(* CoDeSys 2.3.9.42 project: komp_new.pro *)
(* Libraries: Standard.lib 2.12.10 17:48:34, SYSLIBCALLBACK.LIB 2.12.10 17:48:32 *)

(* PLC configuration (modules and I/O channels)
S4_1 AT %IX12.0 [BOOLOnX_I] Ch_1 Digital input
S4_2 AT %IX12.1 [BOOLOnX_I] Ch_2 Digital input
S5_1 AT %IX12.2 [BOOLOnX_I] Ch_3 Digital input
S5_2 AT %IX12.3 [BOOLOnX_I] Ch_4 Digital input
S6_1 AT %IX12.4 [BOOLOnX_I] Ch_5 Digital input
S6_2 AT %IX12.5 [BOOLOnX_I] Ch_6 Digital input
S7_1 AT %IX12.6 [BOOLOnX_I] Ch_7 Digital input
S7_2 AT %IX12.7 [BOOLOnX_I] Ch_8 Digital input
S8_1 AT %IX12.8 [BOOLOnX_I] Ch_9 Digital input
S8_2 AT %IX12.9 [BOOLOnX_I] Ch_10 Digital input
S9_1 AT %IX12.10 [BOOLOnX_I] Ch_11 Digital input
S9_2 AT %IX12.11 [BOOLOnX_I] Ch_12 Digital input
S10_1 AT %IX12.12 [BOOLOnX_I] Ch_13 Digital input
S10_2 AT %IX12.13 [BOOLOnX_I] Ch_14 Digital input
S11_1 AT %IX12.14 [BOOLOnX_I] Ch_15 Digital input
S11_2 AT %IX12.15 [BOOLOnX_I] Ch_16 Digital input
S14_1 AT %IX13.0 [BOOLOnX_I] Ch_1 Digital input
S14_2 AT %IX13.1 [BOOLOnX_I] Ch_2 Digital input
S18_1 AT %IX13.2 [BOOLOnX_I] Ch_3 Digital input
S18_2 AT %IX13.3 [BOOLOnX_I] Ch_4 Digital input
S19_1 AT %IX13.4 [BOOLOnX_I] Ch_5 Digital input
S19_2 AT %IX13.5 [BOOLOnX_I] Ch_6 Digital input
_controlFazaDI AT %IX13.6 [BOOLOnX_I] Ch_7 Digital input
_currentHighJD5DI AT %IX13.7 [BOOLOnX_I] Ch_8 Digital input
_vacumContactOnDI AT %IX13.8 [BOOLOnX_I] Ch_9 Digital input
_vacumContactOffDI AT %IX13.9 [BOOLOnX_I] Ch_10 Digital input
__1pressLevelInDI AT %IX13.10 [BOOLOnX_I] Ch_11 Digital input
__2pressLevelInDI AT %IX13.11 [BOOLOnX_I] Ch_12 Digital input
__3pressLevelInDI AT %IX13.12 [BOOLOnX_I] Ch_13 Digital input
__4pressLevelInDI AT %IX13.13 [BOOLOnX_I] Ch_14 Digital input
_4pressLeveOutDI AT %IX13.14 [BOOLOnX_I] Ch_15 Digital input
pressWaterDI AT %IX13.15 [BOOLOnX_I] Ch_16 Digital input
KM4_1 AT %QX0.0 [BOOLOnX_Q] Ch_1 Digital output
KM4_2 AT %QX0.1 [BOOLOnX_Q] Ch_2 Digital output
KM5_1 AT %QX0.2 [BOOLOnX_Q] Ch_3 Digital output
KM5_2 AT %QX0.3 [BOOLOnX_Q] Ch_4 Digital output
KM6_1 AT %QX0.4 [BOOLOnX_Q] Ch_5 Digital output
KM6_2 AT %QX0.5 [BOOLOnX_Q] Ch_6 Digital output
KM7_1 AT %QX0.6 [BOOLOnX_Q] Ch_7 Digital output
KM7_2 AT %QX0.7 [BOOLOnX_Q] Ch_8 Digital output
KM8_1 AT %QX0.8 [BOOLOnX_Q] Ch_9 Digital output
KM8_2 AT %QX0.9 [BOOLOnX_Q] Ch_10 Digital output
KM9_1 AT %QX0.10 [BOOLOnX_Q] Ch_11 Digital output
KM9_2 AT %QX0.11 [BOOLOnX_Q] Ch_12 Digital output
KM10_1 AT %QX0.12 [BOOLOnX_Q] Ch_13 Digital output
KM10_2 AT %QX0.13 [BOOLOnX_Q] Ch_14 Digital output
KM11_1 AT %QX0.14 [BOOLOnX_Q] Ch_15 Digital output
KM11_2 AT %QX0.15 [BOOLOnX_Q] Ch_16 Digital output
KM14_1 AT %QX1.0 [BOOLOnX_Q] Ch_1 Digital output
KM14_2 AT %QX1.1 [BOOLOnX_Q] Ch_2 Digital output
KM18_1 AT %QX1.2 [BOOLOnX_Q] Ch_3 Digital output
KM18_2 AT %QX1.3 [BOOLOnX_Q] Ch_4 Digital output
readyWater AT %QX1.4 [BOOLOnX_Q] Ch_5 Digital output
readyOil AT %QX1.5 [BOOLOnX_Q] Ch_6 Digital output
_oilGate_1 AT %QX1.6 [BOOLOnX_Q] Ch_7 Digital output
_oilGate_2 AT %QX1.7 [BOOLOnX_Q] Ch_8 Digital output
KM2 AT %QX1.8 [BOOLOnX_Q] Ch_9 Digital output
_rejimModeDO AT %QX1.9 [BOOLOnX_Q] Ch_10 Digital output
KM1 AT %QX1.10 [BOOLOnX_Q] Ch_11 Digital output
_PuskModeDO AT %QX1.11 [BOOLOnX_Q] Ch_12 Digital output
_kompOnDO AT %QX1.12 [BOOLOnX_Q] Ch_13 Digital output
_kompOffDO AT %QX1.13 [BOOLOnX_Q] Ch_14 Digital output
_alarmLedDO_blink AT %QX1.14 [BOOLOnX_Q] Ch_15 Digital output
_stopModeDO AT %QX1.15 [BOOLOnX_Q] Ch_16 Digital output
AT %IW0 [WORDOnW_I] Ch_1 Input word
AT %IW1 [WORDOnW_I] Ch_2 Input word
AT %IW2 [WORDOnW_I] Ch_3 Input word
AT %IW3 [WORDOnW_I] Ch_4 Input word
AT %IW4 [WORDOnW_I] Ch_1 Input word
AT %IW5 [WORDOnW_I] Ch_2 Input word
AT %IW6 [WORDOnW_I] Ch_3 Input word
AT %IW7 [WORDOnW_I] Ch_4 Input word
AT %IW8 [WORDOnW_I] Ch_1 Input word
AT %IW9 [WORDOnW_I] Ch_2 Input word
AT %IW10 [WORDOnW_I] Ch_3 Input word
AT %IW11 [WORDOnW_I] Ch_4 Input word
_konsovikMechanikMotor AT %IX14.0 [BOOLOnX_I] Ch_1 Digital input
_emergencyStop AT %IX14.1 [BOOLOnX_I] Ch_2 Digital input
_buttonStop AT %IX14.2 [BOOLOnX_I] Ch_3 Digital input
_buttonRejim AT %IX14.3 [BOOLOnX_I] Ch_4 Digital input
_buttonPusk AT %IX14.4 [BOOLOnX_I] Ch_5 Digital input
_switchAuto AT %IX14.5 [BOOLOnX_I] Ch_6 Digital input
_switchManual AT %IX14.6 [BOOLOnX_I] Ch_7 Digital input
_emergencyStopMashZal AT %IX14.7 [BOOLOnX_I] Ch_8 Digital input
gazaAnalizMashzal AT %IX14.8 [BOOLOnX_I] Ch_9 Digital input
gazaAnaliz AT %IX14.9 [BOOLOnX_I] Ch_10 Digital input
_pressOilMINDI AT %IX14.10 [BOOLOnX_I] Ch_11 Digital input
_pressOilMAXDI AT %IX14.11 [BOOLOnX_I] Ch_12 Digital input
pressOil_DI AT %IX14.12 [BOOLOnX_I] Ch_13 Digital input
AT %IX14.13 [BOOLOnX_I] Ch_14 Digital input
AT %IX14.14 [BOOLOnX_I] Ch_15 Digital input
AT %IX14.15 [BOOLOnX_I] Ch_16 Digital input
Fieldbus variables [FB_VARS] node 1, in %IB0 out %QB0
Flag variables [FLAG_VARS] node 2, in %IB0 out %QB0
*)

(* Global variable list: _L *)
VAR_GLOBAL
	L11_PUSK : BOOL;
	L12_PUSK : BOOL;
	TO_LIST13: BOOL;

END_VAR

(* Global variable list: _S *)
VAR_GLOBAL
	_17S_1: BOOL;
	_16S_1: BOOL;
END_VAR

(* Global variable list: Global_Variables *)
VAR_GLOBAL
	_alarmLedDO : BOOL;
	alarm : ALARMS;
	_pressWaterDI : BOOL;
	_pressOil_DI : BOOL;
	_1pressLevelInDI : BOOL;
	_2pressLevelInDI : BOOL;
	_3pressLevelInDI : BOOL;
	_4pressLevelInDI : BOOL;
	(*waterPump1 : Pumps;
	waterPump2 : Pumps;
	oilPump1 : Pumps;
	oilPump2 : Pumps;
	_18gate : GateValve;
	_4gate : GateValve;
	_5gate : GateValve;
	_6gate : GateValve;
	_7gate : GateValve;
	_8gate : GateValve;
	_9gate : GateValve;
	_10gate : GateValve;
	_11gate : GateValve;
	_14gate : GateValve;
	_17gate : GateValve;
	_19gate : GateValve;
	_20gate : GateValve;
	heater : Heaters;
	komp : Compressor;

	wtrTimeWORD AT %QW256: WORD := 2;
	oilTimeWORD  AT %QW257: WORD := 2;

	MODE AT %QW280 : WORD;

	gate18TimeWORD  AT %IW258 :WORD := 2;
	gate4TimeWORD  AT %IW259 :WORD := 2;
	gate5TimeWORD  AT %IW260 :WORD := 2;
	gate6TimeWORD  AT %IW261 :WORD := 2;
	gate7TimeWORD  AT %IW262 :WORD := 2;
	gate8TimeWORD  AT %IW263 :WORD := 2;
	gate9TimeWORD  AT %IW264 :WORD := 2;
	gate10TimeWORD  AT %IW265 :WORD := 2;
	gate11TimeWORD  AT %IW266 :WORD := 2;
	gate14TimeWORD  AT %IW267 :WORD := 2;
	gate17TimeWORD  AT %QW268 :WORD := 2;
	gate17T3  AT %IW268 :WORD := 3;
	gate17T4  AT %MW268 :WORD := 4;
	
	wtrTime : TIME := T#2s;
	oilTime : TIME := T#2s;
	gate18Time  :TIME := T#2s;
	gate4Time  :TIME := T#2s;
	gate5Time  :TIME := T#2s;
	gate6Time  :TIME := T#2s;
	gate7Time  :TIME := T#2s;
	gate8Time  :TIME := T#2s;
	gate9Time  :TIME := T#2s;
	gate10Time :TIME := T#2s;
	gate11Time  :TIME := T#2s;
	gate14Time  :TIME := T#2s;
	gate17Time  :TIME := T#2s;

	goRejim AT %QX269.0 : BOOL;
	goPusk AT %QX269.1: BOOL;
	goSTOP AT %QX269.2 : BOOL;
	kompReady AT %QX269.3 : BOOL := FALSE;
	isOK AT %QX269.4: BOOL := TRUE;

	_4gate_open  AT %IX269.5 : BOOL;
	_4gate_close  AT %IX269.6 : BOOL;
	_5gate_open  AT %IX269.7 : BOOL;
	_5gate_close  AT %IX269.8 : BOOL;
	_6gate_open  AT %IX269.9 : BOOL;
	_6gate_close  AT %IX269.10 : BOOL;
	_7gate_open  AT %IX269.11 : BOOL;
	_7gate_close  AT %IX269.12 : BOOL;
	_8gate_open  AT %IX269.13 : BOOL;
	_8gate_close  AT %IX269.14 : BOOL;
	_9gate_open  AT %IX269.15 : BOOL;
	_9gate_close  AT %IX270.0 : BOOL;
	_10gate_open  AT %IX270.1 : BOOL;
	_10gate_close  AT %IX270.2 : BOOL;
	_11gate_open  AT %IX270.3 : BOOL;
	_11gate_close  AT %IX270.4 : BOOL;
	_14gate_open  AT %IX270.5 : BOOL;
	_14gate_close  AT %IX270.6 : BOOL;
	_18gate_open  AT %IX270.7 : BOOL;
	_18gate_close  AT %IX270.8 : BOOL;
	_19gate_open  AT %IX270.9 : BOOL;
	_19gate_close  AT %IX270.10 : BOOL;
	_20gate_open  AT %IX270.11 : BOOL;
	_20gate_close  AT %IX270.12 : BOOL;
	oilPump1_run  AT %IX270.13 : BOOL;
	oilPump2_run  AT %IX270.14 : BOOL;
	waterPump1_run  AT %IX270.15 : BOOL;
	waterPump2_run  AT %IX271.0 : BOOL;
	komp_run  AT %IX271.1 : BOOL;
	komp_stop  AT %IX271.2 : BOOL;
	autoManual  AT %IX272.0 : BOOL;
	*)


END_VAR

(* Global variable list: K *)
VAR_GLOBAL

	K01: BOOL;
	K1: BOOL;
	K2: BOOL;
	K3: BOOL;
	K4: BOOL;
	K5: BOOL;
	K6 : BOOL;
	K7 : BOOL;
	K8 : BOOL;
	K13 : BOOL;
	K14: BOOL;
	K15: BOOL;
END_VAR

(* Global variable list: KM *)
VAR_GLOBAL

	TRM7: BOOL := TRUE;
	KM3: BOOL; (*Nagrev gaza*)
(*
	KM1: BOOL; (* suv nasos*)
	KM2: BOOL; (*maslo nasos*)
	
	KM4_1: BOOL;  (*Zadvijka 4 katushka ochish*)
	KM4_2: BOOL;  (*Zadvijka 4 katushka YOPISH*)
	KM5_1: BOOL;  (*Zadvijka 5 katushka ochish*)
	KM5_2: BOOL;  (*Zadvijka 5 katushka ochish*)
	KM6_1 : BOOL; (*Zadvijka 6 katushka ochish*)
	KM6_2 : BOOL; (*Zadvijka 6 katushka YOPISH*)
	KM7_1: BOOL; (*Zadvijka 7 katushka ochish*)
	KM7_2: BOOL;  (*Zadvijka 7 katushka YOPISH*)
	KM8_1: BOOL; (*Zadvijka 8 katushka ochish*)
	KM8_2: BOOL; (*Zadvijka 8 katushka YOPISH*)
	KM9_1: BOOL;  (*Zadvijka 9 katushka ochish*)
	KM9_2: BOOL;  (*Zadvijka 9 katushka YOPISH*)
	KM10_1: BOOL;  (*Zadvijka 10 katushka ochish*)
	KM10_2: BOOL; (*Zadvijka 10 katushka YOPISH*)
	KM11_1: BOOL; (*Zadvijka 11 katushka ochish*)
	KM11_2: BOOL; (*Zadvijka 11 katushka YOPISH*)
	KM13_1: BOOL;  (*Zadvijka 13 katushka ochish*)
	KM13_2: BOOL; (*Zadvijka 13 katushka YOPISH*)
	KM14_1: BOOL;  (*Zadvijka 14 katushka ochish*)
	KM14_2: BOOL;  (*Zadvijka 14 katushka YOPISH*)
	KM15_1 : BOOL;  (*Zadvijka 15 katushka ochish*)
	KM15_2 : BOOL; (*Zadvijka 15 katushka YOPISH*)
	
	KM18_1 : BOOL; (*Zadvijka 18 katushka ochish*)
	KM18_2 : BOOL;	(*Zadvijka 18 katushka YOPISH*)
*)
	KM16_1: BOOL;  (*Zadvijka 16 katushka ochish*)
	KM16_2: BOOL; (*Zadvijka 16 katushka YOPISH*)
	KM17_1: BOOL; (*Zadvijka 17 katushka ochish*)
	KM17_2: BOOL; (*Zadvijka 17 katushka YOPISH*)
END_VAR

(* Global variable list: P *)
VAR_GLOBAL

	P0: BOOL;

	P1 : BOOL; 	(*GOTOVNOST*)
	P2 : BOOL; 	(*REJIM*)
	P3: BOOL; 	(* STOP kompressor*)
	P4 : BOOL;
	P5 : BOOL;
	P6 : BOOL;	 (* EKM vodinoy nasos*)
	P7 : BOOL; 	(* EKM maslo nasos*)


END_VAR

(* Global variable list: RV *)
VAR_GLOBAL


	RV3: BOOL;
	RV4: BOOL;
	RV5: BOOL;
	RV13: BOOL;
	RV15: BOOL;

	RV3TON: TON;
	RV4TON: TON;
	RV5TON: TON;
	RV13TON : TON;
	RV15TON : TON;


END_VAR

(* Global variable list: V_MODBUS *)
VAR_GLOBAL

	S4_1MB AT %MX100.0 : BOOL;
	S4_2MB AT %MX100.1 : BOOL;
	S5_1MB AT %MX100.2 : BOOL;
	S5_2MB AT %MX100.3 : BOOL;
	S6_1MB AT %MX100.4 : BOOL;
	S6_2MB AT %MX100.5 : BOOL;
	S7_1MB AT %MX100.6 : BOOL;
	S7_2MB AT %MX100.7 : BOOL;
	S8_1MB AT %MX100.8 : BOOL;
	S8_2MB AT %MX100.9 : BOOL;
	S9_1MB AT %MX100.10 : BOOL;
	S9_2MB AT %MX100.11 : BOOL;
	S10_1MB AT %MX100.12 : BOOL;
	S10_2MB AT %MX100.13 : BOOL;
	S11_1MB AT %MX100.14 : BOOL;
	S11_2MB AT %MX100.15 : BOOL;
	S14_1MB AT %MX101.0 : BOOL;
	S14_2MB AT %MX101.1 : BOOL;
	S18_1MB AT %MX101.2 : BOOL;
	S18_2MB AT %MX101.3 : BOOL;
	S19_1MB AT %MX101.4 : BOOL;
	S19_2MB AT %MX101.5 : BOOL;
	controlFazaDIMB AT %MX101.6 : BOOL;
	currentHighJD5DIMB AT %MX101.7 : BOOL;
	vacumContactOnDIMB AT %MX101.8 : BOOL;
	vacumContactOffDIMB AT %MX101.9 : BOOL;
	press1LevelInDIMB AT %MX101.10 : BOOL;
	press2LevelInDIMB AT %MX101.11 : BOOL;
	press3LevelInDIMB AT  %MX101.12 : BOOL;
	press4LevelInDIMB AT %MX101.13 : BOOL;
	press4LevelOutDIMB AT %MX101.14 : BOOL;
	pressWaterDIMB AT  %MX101.15 : BOOL;
	KM4_1MB AT %MX102.0 : BOOL;
	KM4_2MB AT %MX102.1 : BOOL;
	KM5_1MB AT %MX102.2 : BOOL;
	KM5_2MB AT %MX102.3 : BOOL;
	KM6_1MB AT %MX102.4 : BOOL;
	KM6_2MB AT %MX102.5 : BOOL;
	KM7_1MB AT %MX102.6 : BOOL;
	KM7_2MB AT %MX102.7 : BOOL;
	KM8_1MB AT %MX102.8 : BOOL;
	KM8_2MB AT %MX102.9 : BOOL;
	KM9_1MB AT %MX102.10 : BOOL;
	KM9_2MB AT %MX102.11 : BOOL;
	KM10_1MB AT %MX102.12 : BOOL;
	KM10_2MB AT %MX102.13 : BOOL;
	KM11_1MB AT %MX102.14 : BOOL;
	KM11_2MB AT %MX102.15 : BOOL;

	KM14_1MB AT %MX103.0 : BOOL;
	KM14_2MB AT %MX103.1 : BOOL;
	KM18_1MB AT %MX103.2 : BOOL;
	KM18_2MB AT %MX103.3 : BOOL;
	KM19_1MB AT %MX103.4 : BOOL;
	KM19_2MB AT %MX103.5 : BOOL;
	KM1_MB AT %MX103.6 : BOOL;
	KM2_MB AT %MX103.7 : BOOL;
	kompOnDO_MB AT %MX103.8 : BOOL;
	kompOffDO_MB AT %MX103.9 : BOOL;
	alarmLedDO_MB AT %MX103.10 : BOOL;
	stopModeDO_MB AT %MX103.11 : BOOL;
	acknowledgment_MB AT %MX103.12 : BOOL;
	gazaAnaliz_MB AT %MX103.12 : BOOL;
	gazaAnalizMashzal_MB  AT %MX103.13 : BOOL;
	serviceMODE_MB AT %MX103.14 : BOOL;
	SB3 AT %MX104.0: BOOL;  (*PUSK VODA knopka*)
	SB4 AT %MX104.1: BOOL;  (*STOP VODA knopka*)
	SB5 AT %MX104.2: BOOL; (*PUSK MASLO knopka*)
	SB6 AT %MX104.3: BOOL; (*STOP MASLO knopka*)
	SB7 AT %MX104.4: BOOL; (*PUSK NAGREV knopka*)
	SB8 AT %MX104.5: BOOL; (*STOP NAGREV knopka*)
	SB9 AT %MX104.6: BOOL; (*Zadvijka 4 ochish knopka*)
	SB10 AT %MX104.7: BOOL;  (*Zadvijka  4  YOPISH   knopka*)
	SB11 AT %MX104.8: BOOL; (*Zadvijka 5 ochish knopka*)
	SB12 AT %MX104.9: BOOL; (*Zadvijka 5 YOPISH knopka*)
	SB13 AT %MX104.10: BOOL; (*Zadvijka 6 ochish knopka*)
	SB14 AT %MX104.11: BOOL;  (*Zadvijka 6 YOPISH knopka*)
	SB15 AT %MX104.12: BOOL;  (*Zadvijka 7 ochish knopka*)
	SB16 AT %MX104.13: BOOL; (*Zadvijka 7 YOPISH knopka*)
	SB17 AT %MX104.14: BOOL;  (*Zadvijka 8 ochish knopka*)
	SB18 AT %MX104.15: BOOL; (*Zadvijka 8 YOPISH knopka*)

	SB19 AT %MX105.0: BOOL;	 (*Zadvijka 9 ochish knopka*)
	SB20 AT %MX105.1: BOOL;  (*Zadvijka 9 YOPISH knopka*)
	SB21 AT %MX105.2: BOOL;	 (*Zadvijka 10 ochish knopka*)
	SB22 AT %MX105.3: BOOL; (*Zadvijka 10 YOPISH knopka*)
	SB23 AT %MX105.4: BOOL; (*Zadvijka 11 ochish knopka*)
	SB24 AT %MX105.5: BOOL; (*Zadvijka 11 YOPISH knopka*)
	SB25 AT %MX105.6: BOOL;  (*Zadvijka 14 ochish knopka*)
	SB26 AT %MX105.7: BOOL;  (*Zadvijka 14 YOPISH knopka*)
	SB29 AT %MX105.8: BOOL;  (*Zadvijka 18 ochish knopka*)
	SB30 AT %MX105.9: BOOL;   (*Zadvijka 18 YOPISH knopka*)
	SB32 AT %MX105.10: BOOL; (*Zadvijka 16 YOPISH knopka*)
	SBA41 AT %IX14.12: BOOL; (* Avariyniy stop*)
	SBA41_MB AT %MX105.11: BOOL; (* Avariyniy stop*)
	SB42 AT  %IX14.3: BOOL;	 (* knopka REJIM*)
	SB42_MB AT  %MX105.12: BOOL;	 (* knopka REJIM*)
	SB43 AT %IX14.4: BOOL; (* knopka PUSK*)
	SB43_MB AT %MX105.13: BOOL; (* knopka PUSK*)
	SB44 AT %IX14.2: BOOL; (*Kompressor STOP*)
	SB44_MB AT %MX105.14: BOOL; (*Kompressor STOP*)
	(*SB53_1 : BOOL := TRUE; (*obshiy stop zadvijek *)*)
	SB53_1 AT %IX14.2: BOOL; (*obshiy stop zadvijek *)
	SB53_1MB AT %MX105.15 : BOOL; (*obshiy stop zadvijek *)

	(*SBZ AT %IX15.1: BOOL; (*AVARIYNIY STOP MASH ZALA*)*)
	SBZ_MB AT %MX106.0: BOOL; (*AVARIYNIY STOP MASH ZALA*)
	SA45_1MB AT %MX106.1: BOOL;
	SA45_2MB AT %MX106.2: BOOL;
	SB28 : BOOL;  (*Zadvijka 17 YOPISH knopka*)
	SA45_1 : BOOL; (*Auto mode switch*)
	(*SA45_1 AT %IX14.5: BOOL; (*Auto mode switch*)*)
	(*SA45_2 AT %IX14.1: BOOL; (*Emergency stop*)*)
	SA45_2 : BOOL; (*Emergency stop*)



	pressOilMINDI_MB AT %MX107.0 : BOOL;
	rejimModeDO_MB AT  %MX107.1 : BOOL;
	pressOilMAXDI_MB AT %MX107.2 : BOOL;
	puskModeDO_MB AT %MX107.3 :BOOL;
	pressOilDI_MB AT %MX107.4 : BOOL;

	konsovikMechanikMotor AT %MX108.0 : BOOL;
	emergencyStop_MB AT %MX108.1 : BOOL;
	buttonStop_MB AT %MX108.2 : BOOL;
	buttonRejim_MB AT %MX108.3 : BOOL;
	buttonPusk_MB AT %MX108.4 : BOOL;
	switchAuto_MB AT %MX108.5 : BOOL;
	switchManual_MB AT %MX108.6 : BOOL;
	emergencyStopmashZal_MB AT %MX108.7 : BOOL;
	alarrm4levelTemp_MB AT %MX108.8 : BOOL;


	analog1 AT %MW120 : REAL;
	analog2 AT %MW122 : REAL;
	analog3 AT %MW124 : REAL;
	analog4 AT %MW126 : REAL;
	analog5 AT %MW128 : REAL;
	analog6 AT %MW130 : REAL;
	analog7 AT %MW132 : REAL;
	analog8 AT %MW134 : REAL;
	analog9 AT %MW136 : REAL;
	analog10 AT %MW138 : REAL;
	analog11 AT %MW140 : REAL;
	analog12 AT %MW142 : REAL;



END_VAR
VAR_GLOBAL RETAIN PERSISTENT
	analog1SP AT %MW144 : REAL := 250; (*reg 12433*)
	analog2SP AT %MW146 : REAL := 10; (*reg 12435*)
	analog3SP AT %MW148 : REAL := 0.8; (*reg 12437*)
	analog4SP AT %MW150 : REAL := 3.5; (*reg 12439*)

	analog5SP AT %MW152 : REAL := 22; (*reg 12441*)
	analog6SP AT %MW154 : REAL := 64; (*reg 12443*)
	analog7SP AT %MW156 : REAL := 178; (*reg 12445*)
	analog8SP AT %MW158 : REAL := 275; (*reg 12447*)

	analog9SP AT %MW160 : REAL := 1.5; (*reg 12449*)
	analog10SP AT %MW162 : REAL := 150; (*reg 12449*)



END_VAR

(* Data type *)
		TYPE ALARMS :
STRUCT
	gate18NotOpen AT %MX109.0 : BOOL; (* reg 12398.00*)
	gate18NotClose AT %MX109.1 : BOOL; (* reg 12398.01*)

	gate4NotOpen AT %MX109.2 : BOOL; (* reg 12398.02*)
	gate4NotClose AT %MX109.3 : BOOL; (* reg 12398.03*)

	gate5NotOpen AT %MX109.4 : BOOL; (* reg 12398.04*)
	gate5NotClose AT %MX109.5 : BOOL; (* reg 12398.05*)

	gate6NotOpen AT %MX109.6 : BOOL; (* reg 12398.06*)
	gate6NotClose AT %MX109.7 : BOOL; (* reg 12398.07*)

	gate7NotOpen AT %MX109.8 : BOOL; (* reg 12398.08*)
	gate7NotClose AT %MX109.9 : BOOL; (* reg 12398.09*)

	gate8NotOpen AT %MX109.10 : BOOL; (* reg 12398.10*)
	gate8NotClose AT %MX109.11 : BOOL; (* reg 12398.11*)

	gate9NotOpen  AT %MX109.12: BOOL; (* reg 12398.12*)
	gate9NotClose AT %MX109.13 : BOOL; (* reg 12398.13*)

	gate10NotOpen AT %MX109.14 : BOOL; (* reg 12398.14*)
	gate10NotClose AT %MX109.15 : BOOL; (* reg 12398.15*)

	gate11NotOpen AT %MX110.0 : BOOL; (* reg 12399.00*)
	gate11NotClose  AT %MX110.1: BOOL; (* reg 12399.01*)

	gate14NotOpen AT %MX110.2 : BOOL; (* reg 12399.02*)
	gate14NotClose AT %MX110.3 : BOOL; (* reg 12399.03*)
	alarmGazAnaliz AT  %MX110.4 : BOOL; (* reg 12399.04*)
END_STRUCT
END_TYPE

(* POU PLC_PRG, ST *)
PROGRAM PLC_PRG
VAR
END_VAR
SA45_1 := _switchAuto;
SA45_2 := _emergencyStop AND _emergencyStopMashZal ;
translate();
IF (_switchAuto) THEN
	L0005();
	L0008();
	L0009();
	L0010();
	L0011();
	L0012();
	L0013();
	L0014();
	L0015();
	L0016();
END_IF;
gatesAlarm();
start_or_stop();
E_STOP();
blink();
END_PROGRAM

(* POU translate, ST *)
PROGRAM translate
VAR

	K3: BOOL;
	vaqt : TIME := T#2s;
	SC1: SCALE;
	SC2: SCALE;
	SC3: SCALE;
	SC4: SCALE;
	SC5: SCALE;
	SC6: SCALE;
	SC7: SCALE;
	SC8: SCALE;
	SC9: SCALE;
	SC10: SCALE;
	tmrWater : TOF;
	tmrOil: TOF;
	SC11: SCALE;
	SC12: SCALE;
	trig: R_TRIG;
END_VAR
VAR (* helpers for the ST form of the networks *)
	_p1 : BOOL;
END_VAR
MODBUS();
gazaAnaliz_MB := gazaAnaliz;
ANALOG();
ERRORS();
IF (analog1 > analog1SP) THEN
	TRM7 := TRUE;
END_IF;
IF (analog1 < analog1SP - 5) THEN
	TRM7 := FALSE;
END_IF;

K01 := analog3 < analog2SP;
K1 := _1pressLevelInDI;
K2 := _2pressLevelInDI;
K3 := _3pressLevelInDI;
K4 := _4pressLevelInDI;
 _rejimModeDO := (P1 AND _vacumContactOffDI) OR P2;
_stopModeDO := NOT  P1 AND  _vacumContactOffDI;
_PuskModeDO := _vacumContactOnDI;
(*
IF (kompOnDO_MB = TRUE) THEN
	_kompOnDO :=  kompOnDO_MB;
ELSE
	_kompOnDO := FALSE;
END_IF;
IF (kompOffDO_MB = TRUE ) THEN
	_kompOffDO :=  kompOffDO_MB;
ELSE
	_kompOffDO := FALSE;
END_IF
*)
END_PROGRAM
ACTION ANALOG:
		SC1(IN := %IW0, MIN_VALUE := 0, MAX_VALUE := 400, OUT => analog1); (*Akummulator pressure*)
		SC2(IN := %IW1, MIN_VALUE := 0, MAX_VALUE := 400, OUT => analog2); (*Gas pressure 1 level*)
		SC3(IN := %IW2, MIN_VALUE := 0, MAX_VALUE := 400, OUT => analog3);  (*Incomming gas pressure*)
		SC4(IN := %IW3, MIN_VALUE := 0, MAX_VALUE := 400, OUT => analog4);  (*Pressure 2 level*)

		SC5(IN := %IW4,MIN_VALUE := 0, MAX_VALUE := 400,  OUT => analog5); (*Pressure 3 level*)
		SC6(IN := %IW5,MIN_VALUE := 0, MAX_VALUE := 250,  OUT => analog6);     (*Pressure water*)
		SC7(IN := %IW6, MIN_VALUE := 0, MAX_VALUE := 400, OUT => analog7); (*Pressure 4 level*)
		SC8(IN := %IW7, MIN_VALUE := 0, MAX_VALUE := 250, OUT => analog8);   (*Pressure after filtr*)

		SC9(IN := %IW8, MIN_VALUE := 0, MAX_VALUE := 16, OUT => analog9);    (*Pressure before filtr*)
		SC10(IN := %IW9, MIN_VALUE := -50, MAX_VALUE := 150, OUT => analog10); (*Temperture 4 level*)
		SC11(IN := %IW10, MIN_VALUE := -50, MAX_VALUE := 150, OUT => analog11); (*Temperture oil*)
		SC12(IN := %IW11, MIN_VALUE := 0, MAX_VALUE := 1000, OUT => analog12);  (*Motor currency*)
		tmrWater(IN := analog6  > analog3SP, PT := T#5s );
		_pressWaterDI :=  tmrWater.Q;
		readyWater := _pressWaterDI;
		tmrOil(IN := (analog9 > analog4SP AND  analog8 > analog9SP ), PT := T#5s);
		_pressOil_DI    :=  tmrOil.Q;
 		readyOil := _pressOil_DI;

		_1pressLevelInDI    := analog2 >  analog5SP;
		_2pressLevelInDI    := analog4 >  analog6SP;
		_3pressLevelInDI    := analog5 >  analog7SP;
		_4pressLevelInDI    := analog7 >  analog8SP;
		alarrm4levelTemp_MB    := analog10 >  analog10SP;
END_ACTION
ACTION ERRORS:
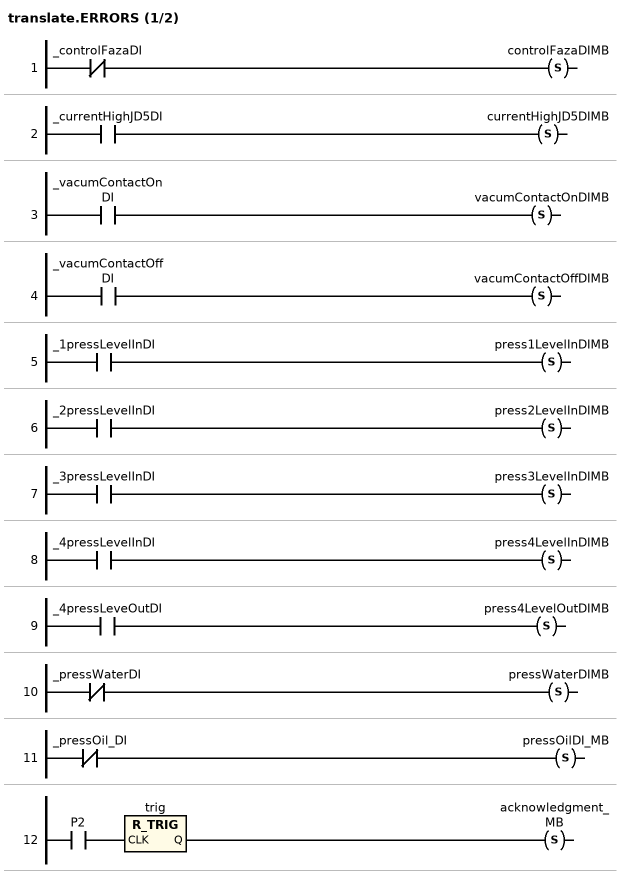
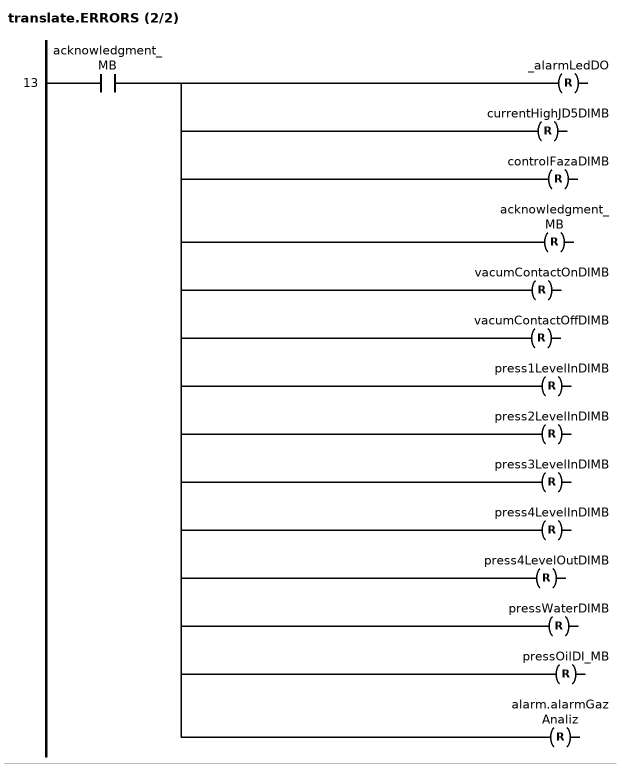
_LD_ (* Ladder Diagram *)
NETWORK 1
	[/_controlFazaDI] --- (S controlFazaDIMB)
NETWORK 2
	[_currentHighJD5DI] --- (S currentHighJD5DIMB)
NETWORK 3
	[_vacumContactOnDI] --- (S vacumContactOnDIMB)
NETWORK 4
	[_vacumContactOffDI] --- (S vacumContactOffDIMB)
NETWORK 5
	[_1pressLevelInDI] --- (S press1LevelInDIMB)
NETWORK 6
	[_2pressLevelInDI] --- (S press2LevelInDIMB)
NETWORK 7
	[_3pressLevelInDI] --- (S press3LevelInDIMB)
NETWORK 8
	[_4pressLevelInDI] --- (S press4LevelInDIMB)
NETWORK 9
	[_4pressLeveOutDI] --- (S press4LevelOutDIMB)
NETWORK 10
	[/_pressWaterDI] --- (S pressWaterDIMB)
NETWORK 11
	[/_pressOil_DI] --- (S pressOilDI_MB)
NETWORK 12
	[P2] - trig:R_TRIG(CLK: *) --- (S acknowledgment_MB)
NETWORK 13
	[acknowledgment_MB] --- (R _alarmLedDO) (R currentHighJD5DIMB) (R controlFazaDIMB) (R acknowledgment_MB) (R vacumContactOnDIMB) (R vacumContactOffDIMB) (R press1LevelInDIMB) (R press2LevelInDIMB) (R press3LevelInDIMB) (R press4LevelInDIMB) (R press4LevelOutDIMB) (R pressWaterDIMB) (R pressOilDI_MB) (R alarm.alarmGazAnaliz)
_END_LD_
(* the same logic as Structured Text *)
(* Network 1 *)
IF NOT _controlFazaDI THEN controlFazaDIMB := TRUE; END_IF;
(* Network 2 *)
IF _currentHighJD5DI THEN currentHighJD5DIMB := TRUE; END_IF;
(* Network 3 *)
IF _vacumContactOnDI THEN vacumContactOnDIMB := TRUE; END_IF;
(* Network 4 *)
IF _vacumContactOffDI THEN vacumContactOffDIMB := TRUE; END_IF;
(* Network 5 *)
IF _1pressLevelInDI THEN press1LevelInDIMB := TRUE; END_IF;
(* Network 6 *)
IF _2pressLevelInDI THEN press2LevelInDIMB := TRUE; END_IF;
(* Network 7 *)
IF _3pressLevelInDI THEN press3LevelInDIMB := TRUE; END_IF;
(* Network 8 *)
IF _4pressLevelInDI THEN press4LevelInDIMB := TRUE; END_IF;
(* Network 9 *)
IF _4pressLeveOutDI THEN press4LevelOutDIMB := TRUE; END_IF;
(* Network 10 *)
IF NOT _pressWaterDI THEN pressWaterDIMB := TRUE; END_IF;
(* Network 11 *)
IF NOT _pressOil_DI THEN pressOilDI_MB := TRUE; END_IF;
(* Network 12 *)
trig(CLK := P2);
IF trig.Q THEN acknowledgment_MB := TRUE; END_IF;
(* Network 13 *)
_p1 := acknowledgment_MB;
IF _p1 THEN _alarmLedDO := FALSE; currentHighJD5DIMB := FALSE; controlFazaDIMB := FALSE; acknowledgment_MB := FALSE; vacumContactOnDIMB := FALSE; vacumContactOffDIMB := FALSE; press1LevelInDIMB := FALSE; press2LevelInDIMB := FALSE; press3LevelInDIMB := FALSE; press4LevelInDIMB := FALSE; press4LevelOutDIMB := FALSE; pressWaterDIMB := FALSE; pressOilDI_MB := FALSE; alarm.alarmGazAnaliz := FALSE; END_IF;
END_ACTION
ACTION MODBUS:
S4_1MB := S4_1;
S4_2MB := S4_2;
S5_1MB := S5_1;
S5_2MB := S5_2;
S6_1MB := S6_1;
S6_2MB := S6_2;
S7_1MB := S7_1;
S7_2MB := S7_2;
S8_1MB := S8_1;
S8_2MB := S8_2;
S9_1MB := S9_1;
S9_2MB := S9_2;
S10_1MB := S10_1;
S10_2MB := S10_2;
S11_1MB := S11_1;
S11_2MB := S11_2;
S14_1MB := S14_1;
S14_2MB := S14_2;
S18_1MB := S18_1;
S18_2MB := S18_2;
S19_1MB := S19_1;
S19_2MB := S19_2;


KM4_1MB := KM4_1;
KM4_2MB := KM4_2;
KM5_1MB := KM5_1;
KM5_2MB := KM5_2;
KM6_1MB := KM6_1;
KM6_2MB := KM6_2;
KM7_1MB := KM7_1;
KM7_2MB := KM7_2;
KM8_1MB := KM8_1;
KM8_2MB := KM8_2;
KM9_1MB := KM9_1;
KM9_2MB := KM9_2;
KM10_1MB := KM10_1;
KM10_2MB := KM10_2;
KM11_1MB := KM11_1;
KM11_2MB := KM11_2;

KM14_1MB := KM14_1;
KM14_2MB := KM14_2;
KM18_1MB := KM18_1;
KM18_2MB := KM18_2;
KM19_1MB := _oilGate_1;
KM19_2MB := _oilGate_2;
KM1_MB := KM1;
KM2_MB := KM2;
(*
kompOnDO_MB := _kompOnDO;
kompOffDO_MB := _kompOffDO;*)
alarmLedDO_MB := _alarmLedDO;
stopModeDO_MB := _stopModeDO;

konsovikMechanikMotor := _konsovikMechanikMotor;
emergencyStop_MB := NOT _emergencyStop;
SBA41_MB := SBA41;
SB42_MB := SB42;
SB43_MB := SB43;
SB44_MB := SB44;
SB53_1MB := SB53_1;




buttonStop_MB := _buttonStop;
buttonRejim_MB := _buttonRejim;
buttonPusk_MB := _buttonPusk;
switchAuto_MB := _switchAuto;
switchManual_MB := _switchManual;
emergencyStopmashZal_MB := NOT  _emergencyStopMashZal;
END_ACTION

(* POU SCALE, ST *)
FUNCTION_BLOCK SCALE
VAR_INPUT
	IN : WORD;
	MIN_VALUE : REAL := 4;
	MAX_VALUE : REAL := 20;
END_VAR
VAR_OUTPUT
	OUT : REAL;
END_VAR
VAR
	T : REAL;
	t2 : REAL;
	n : INT := 0;
	tp1 : TP;
	reset :BOOL;
	vaqt : TIME  := T#300ms;
END_VAR
T := WORD_TO_REAL(IN);
tp1(in := reset, PT := vaqt);
IF (tp1.Q) THEN
	n := n + 1;
	T2 := T2 +  (MAX_VALUE - MIN_VALUE) * T / 32767 +  MIN_VALUE;
ELSE
	out := T2 / n;
	n := 0;
	T2 := 0;
END_IF;
reset := NOT tp1.Q;
END_FUNCTION_BLOCK

(* POU alarm, CFC *)
FUNCTION_BLOCK alarm
VAR_INPUT
	start : BOOL;
	vaqtSekund : WORD := 45;
	konsevik : BOOL;
END_VAR
VAR_OUTPUT
	out : BOOL;
END_VAR
VAR
	TP: TON;
	temp: BOOL;
	rtrig: R_TRIG;
END_VAR
VAR (* helpers for the ST form of the networks *)
	_t8 : BOOL;
	_t4 : TIME;
END_VAR
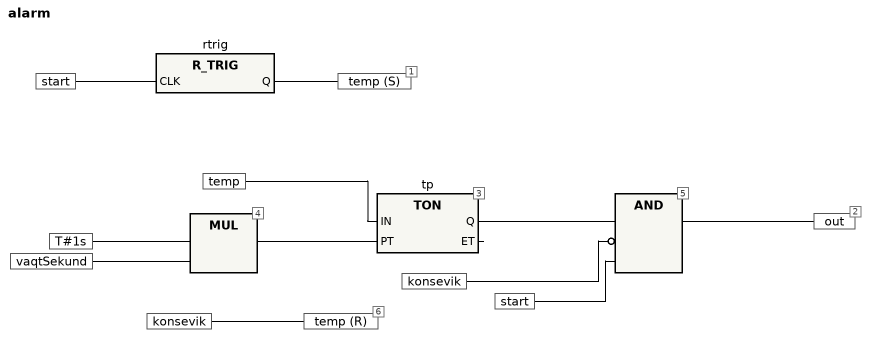
_CFC_ (* Continuous Function Chart, elements in execution order *)
#0 rtrig:R_TRIG(CLK: start)
#1 S temp <= #0.Q
#2 out <= #5
#3 tp:TON(IN: temp, PT: #4)
#4 MUL(T#1s, vaqtSekund)
#5 AND(#3.Q, NOT konsevik, start)
#6 R temp <= konsevik
_END_CFC_
(* the same logic as Structured Text *)
rtrig(CLK := start);
IF rtrig.Q THEN temp := TRUE; END_IF;
out := _t8;
tp(IN := temp, PT := _t4);
_t4 := T#1s * vaqtSekund;
_t8 := tp.Q AND NOT konsevik AND start;
IF konsevik THEN temp := FALSE; END_IF;
END_FUNCTION_BLOCK

(* POU L0005, LD *)
PROGRAM L0005
VAR
	_kompOffDO000000000: BOOL;
	t6AfterTON : TON;

END_VAR
VAR
	_ImpVar_52_3:	BOOL;
	_ImpVar_52_5:	BOOL;
	_ImpVar_52_6:	BOOL;
	_ImpVar_52_14:	BOOL;
	_ImpVar_52_13:	BOOL;
	_ImpVar_52_20:	BOOL;
	_ImpVar_52_21:	BOOL;
	_ImpVar_52_36:	BOOL;
	_ImpVar_52_121:	BOOL;
	_ImpVar_52_46:	BOOL;
	_ImpVar_52_50:	BOOL;
	_ImpVar_52_141:	BOOL;
	_ImpVar_52_57:	BOOL;

END_VAR
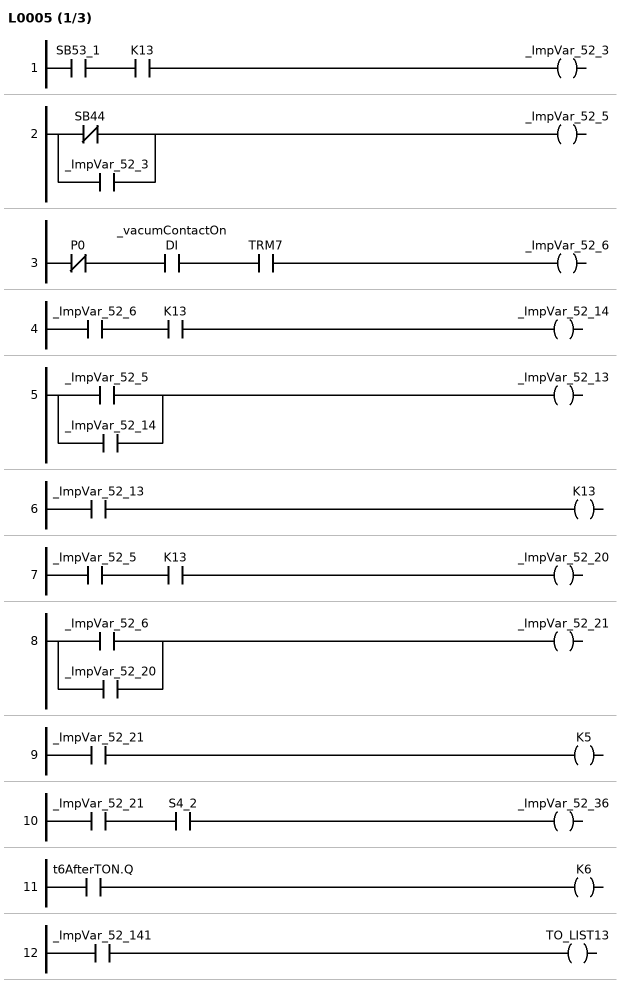
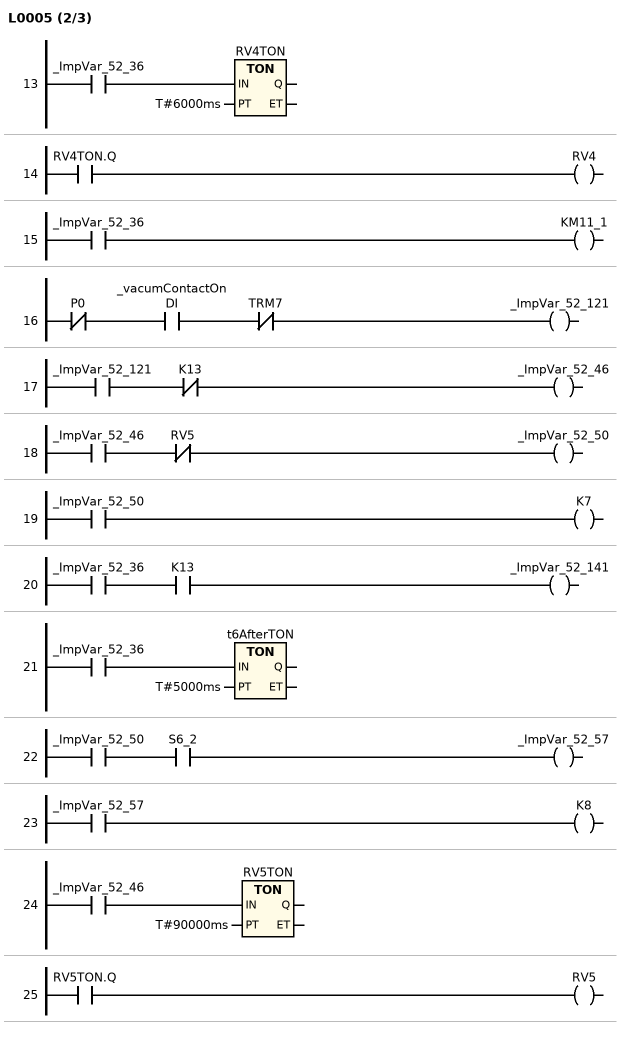
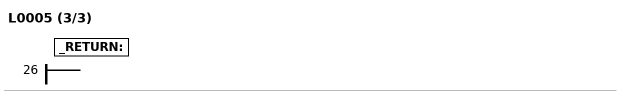
_LD_ (* Ladder Diagram *)
NETWORK 1
	[SB53_1] - [K13] --- (_ImpVar_52_3)
NETWORK 2
	{ [/SB44] | [_ImpVar_52_3] } --- (_ImpVar_52_5)
NETWORK 3
	[/P0] - [_vacumContactOnDI] - [TRM7] --- (_ImpVar_52_6)
NETWORK 4
	[_ImpVar_52_6] - [K13] --- (_ImpVar_52_14)
NETWORK 5
	{ [_ImpVar_52_5] | [_ImpVar_52_14] } --- (_ImpVar_52_13)
NETWORK 6
	[_ImpVar_52_13] --- (K13)
NETWORK 7
	[_ImpVar_52_5] - [K13] --- (_ImpVar_52_20)
NETWORK 8
	{ [_ImpVar_52_6] | [_ImpVar_52_20] } --- (_ImpVar_52_21)
NETWORK 9
	[_ImpVar_52_21] --- (K5)
NETWORK 10
	[_ImpVar_52_21] - [S4_2] --- (_ImpVar_52_36)
NETWORK 11
	[t6AfterTON.Q] --- (K6)
NETWORK 12
	[_ImpVar_52_141] --- (TO_LIST13)
NETWORK 13
	[_ImpVar_52_36] - RV4TON:TON(IN: *, PT: T#6000ms)
NETWORK 14
	[RV4TON.Q] --- (RV4)
NETWORK 15
	[_ImpVar_52_36] --- (KM11_1)
NETWORK 16
	[/P0] - [_vacumContactOnDI] - [/TRM7] --- (_ImpVar_52_121)
NETWORK 17
	[_ImpVar_52_121] - [/K13] --- (_ImpVar_52_46)
NETWORK 18
	[_ImpVar_52_46] - [/RV5] --- (_ImpVar_52_50)
NETWORK 19
	[_ImpVar_52_50] --- (K7)
NETWORK 20
	[_ImpVar_52_36] - [K13] --- (_ImpVar_52_141)
NETWORK 21
	[_ImpVar_52_36] - t6AfterTON:TON(IN: *, PT: T#5000ms)
NETWORK 22
	[_ImpVar_52_50] - [S6_2] --- (_ImpVar_52_57)
NETWORK 23
	[_ImpVar_52_57] --- (K8)
NETWORK 24
	[_ImpVar_52_46] - RV5TON:TON(IN: *, PT: T#90000ms)
NETWORK 25
	[RV5TON.Q] --- (RV5)
NETWORK 26 _RETURN::
	*
_END_LD_
(* the same logic as Structured Text *)
(* Network 1 *)
_ImpVar_52_3 := SB53_1 AND K13;
(* Network 2 *)
_ImpVar_52_5 := NOT SB44 OR _ImpVar_52_3;
(* Network 3 *)
_ImpVar_52_6 := NOT P0 AND _vacumContactOnDI AND TRM7;
(* Network 4 *)
_ImpVar_52_14 := _ImpVar_52_6 AND K13;
(* Network 5 *)
_ImpVar_52_13 := _ImpVar_52_5 OR _ImpVar_52_14;
(* Network 6 *)
K13 := _ImpVar_52_13;
(* Network 7 *)
_ImpVar_52_20 := _ImpVar_52_5 AND K13;
(* Network 8 *)
_ImpVar_52_21 := _ImpVar_52_6 OR _ImpVar_52_20;
(* Network 9 *)
K5 := _ImpVar_52_21;
(* Network 10 *)
_ImpVar_52_36 := _ImpVar_52_21 AND S4_2;
(* Network 11 *)
K6 := t6AfterTON.Q;
(* Network 12 *)
TO_LIST13 := _ImpVar_52_141;
(* Network 13 *)
RV4TON(IN := _ImpVar_52_36, PT := T#6000ms);
(* Network 14 *)
RV4 := RV4TON.Q;
(* Network 15 *)
KM11_1 := _ImpVar_52_36;
(* Network 16 *)
_ImpVar_52_121 := NOT P0 AND _vacumContactOnDI AND NOT TRM7;
(* Network 17 *)
_ImpVar_52_46 := _ImpVar_52_121 AND NOT K13;
(* Network 18 *)
_ImpVar_52_50 := _ImpVar_52_46 AND NOT RV5;
(* Network 19 *)
K7 := _ImpVar_52_50;
(* Network 20 *)
_ImpVar_52_141 := _ImpVar_52_36 AND K13;
(* Network 21 *)
t6AfterTON(IN := _ImpVar_52_36, PT := T#5000ms);
(* Network 22 *)
_ImpVar_52_57 := _ImpVar_52_50 AND S6_2;
(* Network 23 *)
K8 := _ImpVar_52_57;
(* Network 24 *)
RV5TON(IN := _ImpVar_52_46, PT := T#90000ms);
(* Network 25 *)
RV5 := RV5TON.Q;
(* Network 26 *)
(* label: _RETURN: *)
END_PROGRAM

(* POU L0008, LD *)
PROGRAM L0008
VAR


END_VAR
VAR
	_ImpVar_54_53:	BOOL;
	_ImpVar_54_2:	BOOL;
	_ImpVar_54_84:	BOOL;
	_ImpVar_54_27:	BOOL;

END_VAR
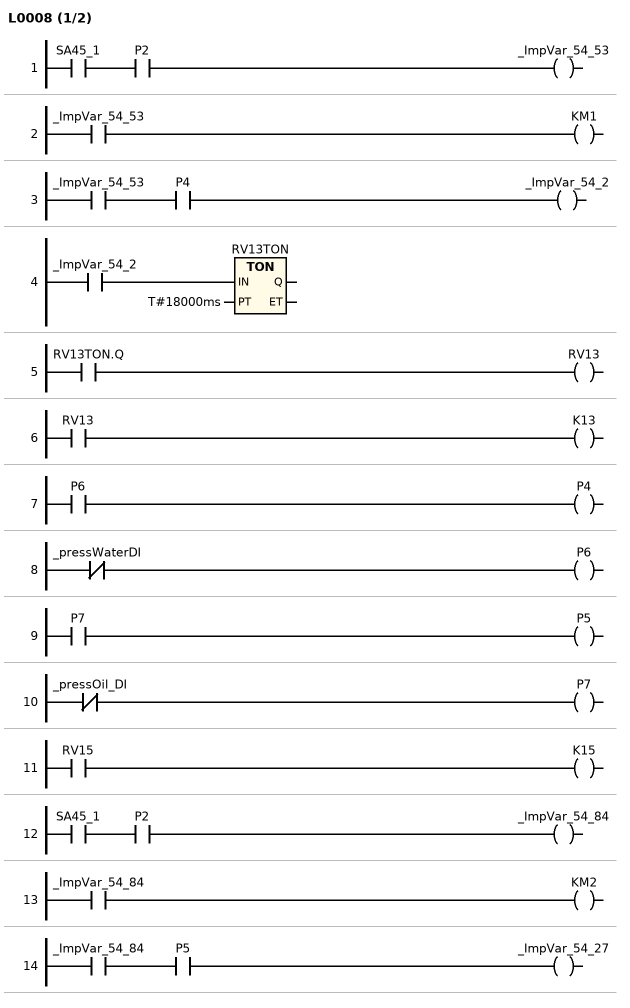
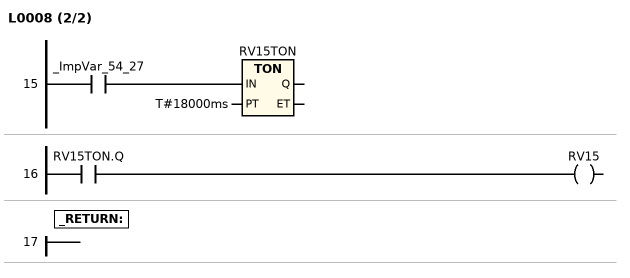
_LD_ (* Ladder Diagram *)
NETWORK 1
	[SA45_1] - [P2] --- (_ImpVar_54_53)
NETWORK 2
	[_ImpVar_54_53] --- (KM1)
NETWORK 3
	[_ImpVar_54_53] - [P4] --- (_ImpVar_54_2)
NETWORK 4
	[_ImpVar_54_2] - RV13TON:TON(IN: *, PT: T#18000ms)
NETWORK 5
	[RV13TON.Q] --- (RV13)
NETWORK 6
	[RV13] --- (K13)
NETWORK 7
	[P6] --- (P4)
NETWORK 8
	[/_pressWaterDI] --- (P6)
NETWORK 9
	[P7] --- (P5)
NETWORK 10
	[/_pressOil_DI] --- (P7)
NETWORK 11
	[RV15] --- (K15)
NETWORK 12
	[SA45_1] - [P2] --- (_ImpVar_54_84)
NETWORK 13
	[_ImpVar_54_84] --- (KM2)
NETWORK 14
	[_ImpVar_54_84] - [P5] --- (_ImpVar_54_27)
NETWORK 15
	[_ImpVar_54_27] - RV15TON:TON(IN: *, PT: T#18000ms)
NETWORK 16
	[RV15TON.Q] --- (RV15)
NETWORK 17 _RETURN::
	*
_END_LD_
(* the same logic as Structured Text *)
(* Network 1 *)
_ImpVar_54_53 := SA45_1 AND P2;
(* Network 2 *)
KM1 := _ImpVar_54_53;
(* Network 3 *)
_ImpVar_54_2 := _ImpVar_54_53 AND P4;
(* Network 4 *)
RV13TON(IN := _ImpVar_54_2, PT := T#18000ms);
(* Network 5 *)
RV13 := RV13TON.Q;
(* Network 6 *)
K13 := RV13;
(* Network 7 *)
P4 := P6;
(* Network 8 *)
P6 := NOT _pressWaterDI;
(* Network 9 *)
P5 := P7;
(* Network 10 *)
P7 := NOT _pressOil_DI;
(* Network 11 *)
K15 := RV15;
(* Network 12 *)
_ImpVar_54_84 := SA45_1 AND P2;
(* Network 13 *)
KM2 := _ImpVar_54_84;
(* Network 14 *)
_ImpVar_54_27 := _ImpVar_54_84 AND P5;
(* Network 15 *)
RV15TON(IN := _ImpVar_54_27, PT := T#18000ms);
(* Network 16 *)
RV15 := RV15TON.Q;
(* Network 17 *)
(* label: _RETURN: *)
END_PROGRAM

(* POU L0009, LD *)
PROGRAM L0009
VAR




	S18_1_prymoy: BOOL := TRUE;
END_VAR
VAR
	_ImpVar_61_2:	BOOL;
	_ImpVar_61_5:	BOOL;
	_ImpVar_61_9:	BOOL;
	_ImpVar_61_49:	BOOL;
	_ImpVar_61_13:	BOOL;
	_ImpVar_61_37:	BOOL;
	_ImpVar_61_23:	BOOL;
	_ImpVar_61_38:	BOOL;
	_ImpVar_61_35:	BOOL;
	_ImpVar_61_40:	BOOL;
	_ImpVar_61_26:	BOOL;
	_ImpVar_61_29:	BOOL;

END_VAR
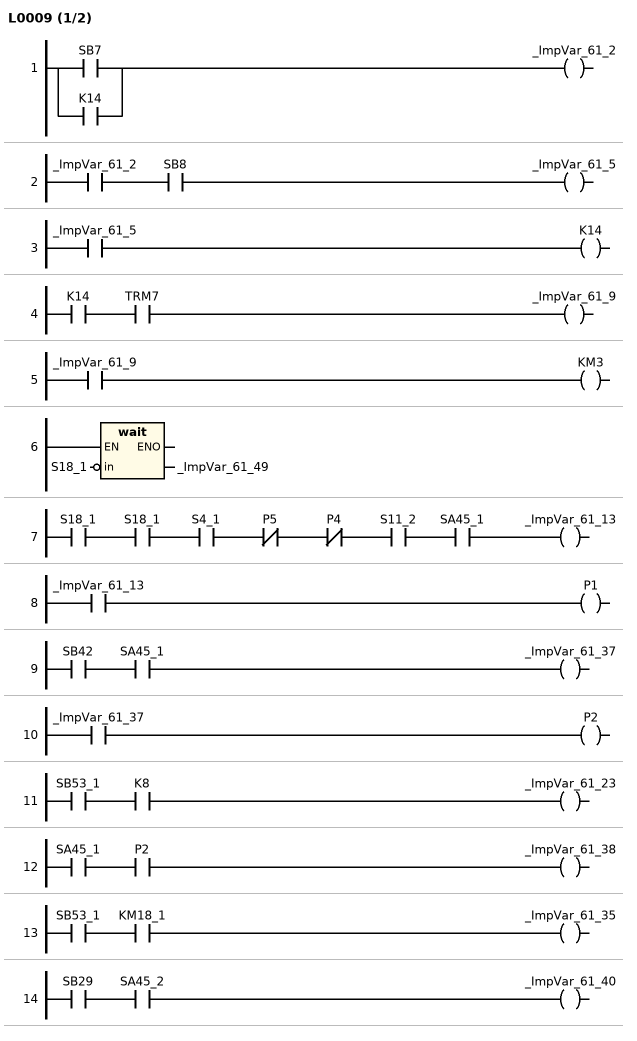
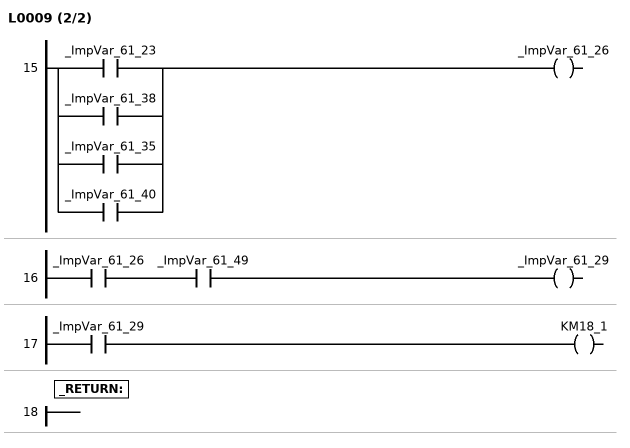
_LD_ (* Ladder Diagram *)
NETWORK 1
	{ [SB7] | [K14] } --- (_ImpVar_61_2)
NETWORK 2
	[_ImpVar_61_2] - [SB8] --- (_ImpVar_61_5)
NETWORK 3
	[_ImpVar_61_5] --- (K14)
NETWORK 4
	[K14] - [TRM7] --- (_ImpVar_61_9)
NETWORK 5
	[_ImpVar_61_9] --- (KM3)
NETWORK 6
	*
		EN --- wait(in: NOT S18_1) => _ImpVar_61_49
NETWORK 7
	[S18_1] - [S18_1] - [S4_1] - [/P5] - [/P4] - [S11_2] - [SA45_1] --- (_ImpVar_61_13)
NETWORK 8
	[_ImpVar_61_13] --- (P1)
NETWORK 9
	[SB42] - [SA45_1] --- (_ImpVar_61_37)
NETWORK 10
	[_ImpVar_61_37] --- (P2)
NETWORK 11
	[SB53_1] - [K8] --- (_ImpVar_61_23)
NETWORK 12
	[SA45_1] - [P2] --- (_ImpVar_61_38)
NETWORK 13
	[SB53_1] - [KM18_1] --- (_ImpVar_61_35)
NETWORK 14
	[SB29] - [SA45_2] --- (_ImpVar_61_40)
NETWORK 15
	{ [_ImpVar_61_23] | [_ImpVar_61_38] | [_ImpVar_61_35] | [_ImpVar_61_40] } --- (_ImpVar_61_26)
NETWORK 16
	[_ImpVar_61_26] - [_ImpVar_61_49] --- (_ImpVar_61_29)
NETWORK 17
	[_ImpVar_61_29] --- (KM18_1)
NETWORK 18 _RETURN::
	*
_END_LD_
(* the same logic as Structured Text *)
(* Network 1 *)
_ImpVar_61_2 := SB7 OR K14;
(* Network 2 *)
_ImpVar_61_5 := _ImpVar_61_2 AND SB8;
(* Network 3 *)
K14 := _ImpVar_61_5;
(* Network 4 *)
_ImpVar_61_9 := K14 AND TRM7;
(* Network 5 *)
KM3 := _ImpVar_61_9;
(* Network 6 *)
_ImpVar_61_49 := wait(in := NOT S18_1);
(* Network 7 *)
_ImpVar_61_13 := S18_1 AND S18_1 AND S4_1 AND NOT P5 AND NOT P4 AND S11_2 AND SA45_1;
(* Network 8 *)
P1 := _ImpVar_61_13;
(* Network 9 *)
_ImpVar_61_37 := SB42 AND SA45_1;
(* Network 10 *)
P2 := _ImpVar_61_37;
(* Network 11 *)
_ImpVar_61_23 := SB53_1 AND K8;
(* Network 12 *)
_ImpVar_61_38 := SA45_1 AND P2;
(* Network 13 *)
_ImpVar_61_35 := SB53_1 AND KM18_1;
(* Network 14 *)
_ImpVar_61_40 := SB29 AND SA45_2;
(* Network 15 *)
_ImpVar_61_26 := _ImpVar_61_23 OR _ImpVar_61_38 OR _ImpVar_61_35 OR _ImpVar_61_40;
(* Network 16 *)
_ImpVar_61_29 := _ImpVar_61_26 AND _ImpVar_61_49;
(* Network 17 *)
KM18_1 := _ImpVar_61_29;
(* Network 18 *)
(* label: _RETURN: *)
END_PROGRAM

(* POU wait, LD *)
FUNCTION wait : BOOL
VAR_INPUT
	in : BOOL;
END_VAR
VAR
	vaqt : TIME := T#120s;
	tp1: TOF;
END_VAR
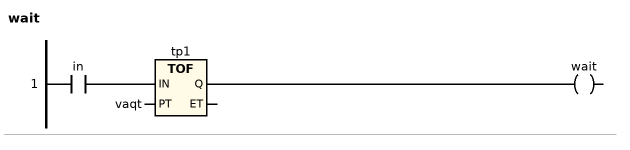
_LD_ (* Ladder Diagram *)
NETWORK 1
	[in] - tp1:TOF(IN: *, PT: vaqt) --- (wait)
_END_LD_
(* the same logic as Structured Text *)
(* Network 1 *)
tp1(IN := in, PT := vaqt);
wait := tp1.Q;
END_FUNCTION

(* POU L0010, LD *)
PROGRAM L0010
VAR
	_17S_2: BOOL;

END_VAR
VAR
	_ImpVar_64_67:	BOOL;
	_ImpVar_64_27:	BOOL;
	_ImpVar_64_2:	BOOL;
	_ImpVar_64_4:	BOOL;
	_ImpVar_64_8:	BOOL;
	_ImpVar_64_9:	BOOL;
	_ImpVar_64_14:	BOOL;
	_ImpVar_64_17:	BOOL;
	_ImpVar_64_29:	BOOL;
	_ImpVar_64_20:	BOOL;
	_ImpVar_64_21:	BOOL;
	_ImpVar_64_30:	BOOL;
	_ImpVar_64_37:	BOOL;
	_ImpVar_64_35:	BOOL;
	_ImpVar_64_32:	BOOL;
	_ImpVar_64_40:	BOOL;
	_ImpVar_64_41:	BOOL;
	_ImpVar_64_68:	BOOL;
	_ImpVar_64_69:	BOOL;

END_VAR
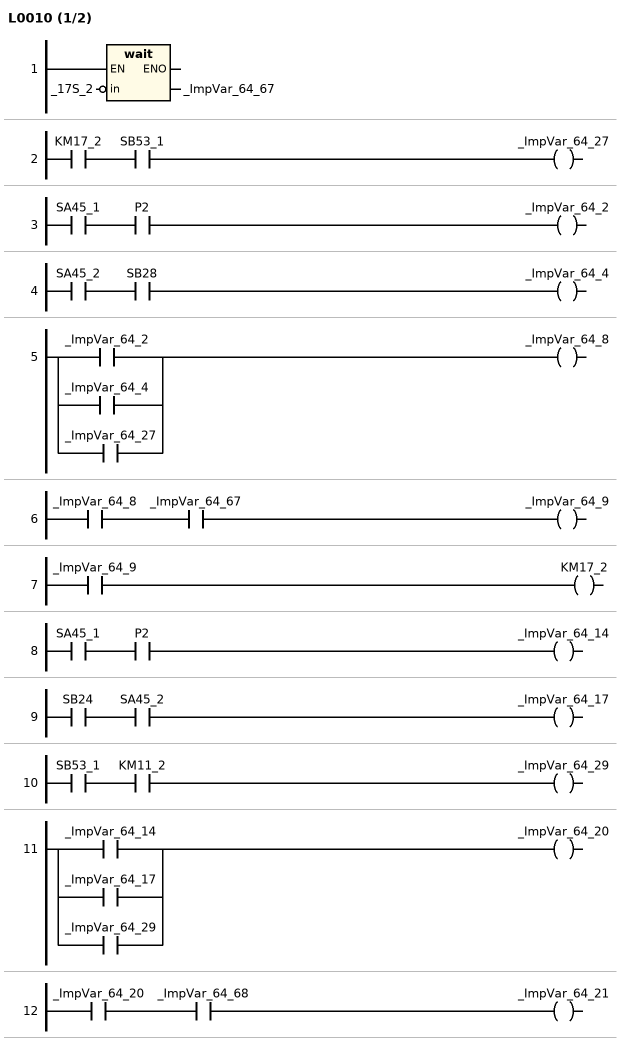
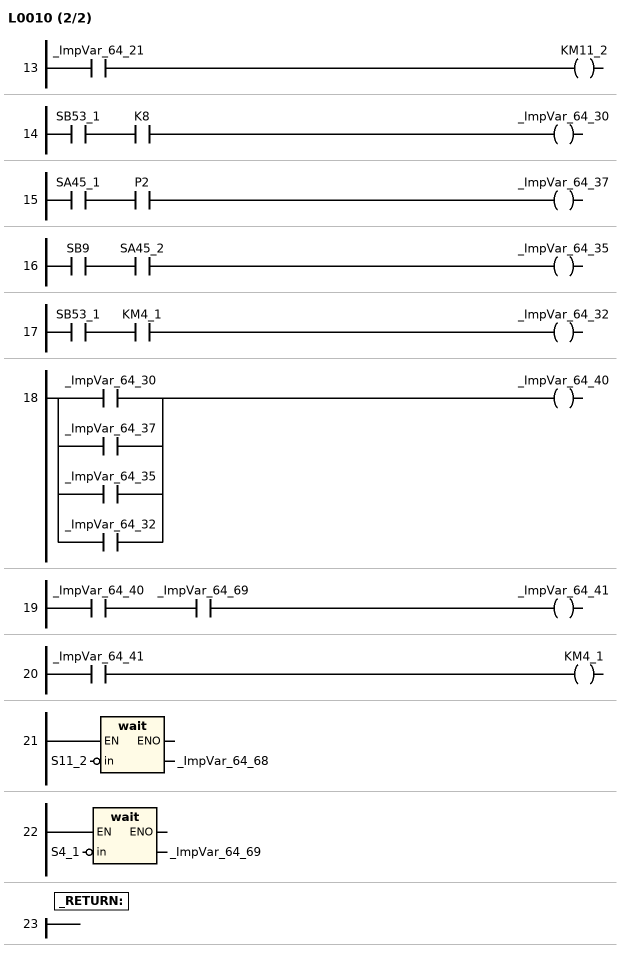
_LD_ (* Ladder Diagram *)
NETWORK 1
	*
		EN --- wait(in: NOT _17S_2) => _ImpVar_64_67
NETWORK 2
	[KM17_2] - [SB53_1] --- (_ImpVar_64_27)
NETWORK 3
	[SA45_1] - [P2] --- (_ImpVar_64_2)
NETWORK 4
	[SA45_2] - [SB28] --- (_ImpVar_64_4)
NETWORK 5
	{ [_ImpVar_64_2] | [_ImpVar_64_4] | [_ImpVar_64_27] } --- (_ImpVar_64_8)
NETWORK 6
	[_ImpVar_64_8] - [_ImpVar_64_67] --- (_ImpVar_64_9)
NETWORK 7
	[_ImpVar_64_9] --- (KM17_2)
NETWORK 8
	[SA45_1] - [P2] --- (_ImpVar_64_14)
NETWORK 9
	[SB24] - [SA45_2] --- (_ImpVar_64_17)
NETWORK 10
	[SB53_1] - [KM11_2] --- (_ImpVar_64_29)
NETWORK 11
	{ [_ImpVar_64_14] | [_ImpVar_64_17] | [_ImpVar_64_29] } --- (_ImpVar_64_20)
NETWORK 12
	[_ImpVar_64_20] - [_ImpVar_64_68] --- (_ImpVar_64_21)
NETWORK 13
	[_ImpVar_64_21] --- (KM11_2)
NETWORK 14
	[SB53_1] - [K8] --- (_ImpVar_64_30)
NETWORK 15
	[SA45_1] - [P2] --- (_ImpVar_64_37)
NETWORK 16
	[SB9] - [SA45_2] --- (_ImpVar_64_35)
NETWORK 17
	[SB53_1] - [KM4_1] --- (_ImpVar_64_32)
NETWORK 18
	{ [_ImpVar_64_30] | [_ImpVar_64_37] | [_ImpVar_64_35] | [_ImpVar_64_32] } --- (_ImpVar_64_40)
NETWORK 19
	[_ImpVar_64_40] - [_ImpVar_64_69] --- (_ImpVar_64_41)
NETWORK 20
	[_ImpVar_64_41] --- (KM4_1)
NETWORK 21
	*
		EN --- wait(in: NOT S11_2) => _ImpVar_64_68
NETWORK 22
	*
		EN --- wait(in: NOT S4_1) => _ImpVar_64_69
NETWORK 23 _RETURN::
	*
_END_LD_
(* the same logic as Structured Text *)
(* Network 1 *)
_ImpVar_64_67 := wait(in := NOT _17S_2);
(* Network 2 *)
_ImpVar_64_27 := KM17_2 AND SB53_1;
(* Network 3 *)
_ImpVar_64_2 := SA45_1 AND P2;
(* Network 4 *)
_ImpVar_64_4 := SA45_2 AND SB28;
(* Network 5 *)
_ImpVar_64_8 := _ImpVar_64_2 OR _ImpVar_64_4 OR _ImpVar_64_27;
(* Network 6 *)
_ImpVar_64_9 := _ImpVar_64_8 AND _ImpVar_64_67;
(* Network 7 *)
KM17_2 := _ImpVar_64_9;
(* Network 8 *)
_ImpVar_64_14 := SA45_1 AND P2;
(* Network 9 *)
_ImpVar_64_17 := SB24 AND SA45_2;
(* Network 10 *)
_ImpVar_64_29 := SB53_1 AND KM11_2;
(* Network 11 *)
_ImpVar_64_20 := _ImpVar_64_14 OR _ImpVar_64_17 OR _ImpVar_64_29;
(* Network 12 *)
_ImpVar_64_21 := _ImpVar_64_20 AND _ImpVar_64_68;
(* Network 13 *)
KM11_2 := _ImpVar_64_21;
(* Network 14 *)
_ImpVar_64_30 := SB53_1 AND K8;
(* Network 15 *)
_ImpVar_64_37 := SA45_1 AND P2;
(* Network 16 *)
_ImpVar_64_35 := SB9 AND SA45_2;
(* Network 17 *)
_ImpVar_64_32 := SB53_1 AND KM4_1;
(* Network 18 *)
_ImpVar_64_40 := _ImpVar_64_30 OR _ImpVar_64_37 OR _ImpVar_64_35 OR _ImpVar_64_32;
(* Network 19 *)
_ImpVar_64_41 := _ImpVar_64_40 AND _ImpVar_64_69;
(* Network 20 *)
KM4_1 := _ImpVar_64_41;
(* Network 21 *)
_ImpVar_64_68 := wait(in := NOT S11_2);
(* Network 22 *)
_ImpVar_64_69 := wait(in := NOT S4_1);
(* Network 23 *)
(* label: _RETURN: *)
END_PROGRAM

(* POU L0011, LD *)
PROGRAM L0011
VAR


	_16S_2: BOOL;
END_VAR
VAR
	_ImpVar_68_2:	BOOL;
	_ImpVar_68_4:	BOOL;
	_ImpVar_68_7:	BOOL;
	_ImpVar_68_10:	BOOL;
	_ImpVar_68_11:	BOOL;
	_ImpVar_68_17:	BOOL;
	_ImpVar_68_21:	BOOL;
	_ImpVar_68_23:	BOOL;
	_ImpVar_68_25:	BOOL;
	_ImpVar_68_26:	BOOL;
	_ImpVar_68_31:	BOOL;
	_ImpVar_68_34:	BOOL;
	_ImpVar_68_36:	BOOL;
	_ImpVar_68_38:	BOOL;
	_ImpVar_68_44:	BOOL;
	_ImpVar_68_54:	BOOL;
	_ImpVar_68_55:	BOOL;

END_VAR
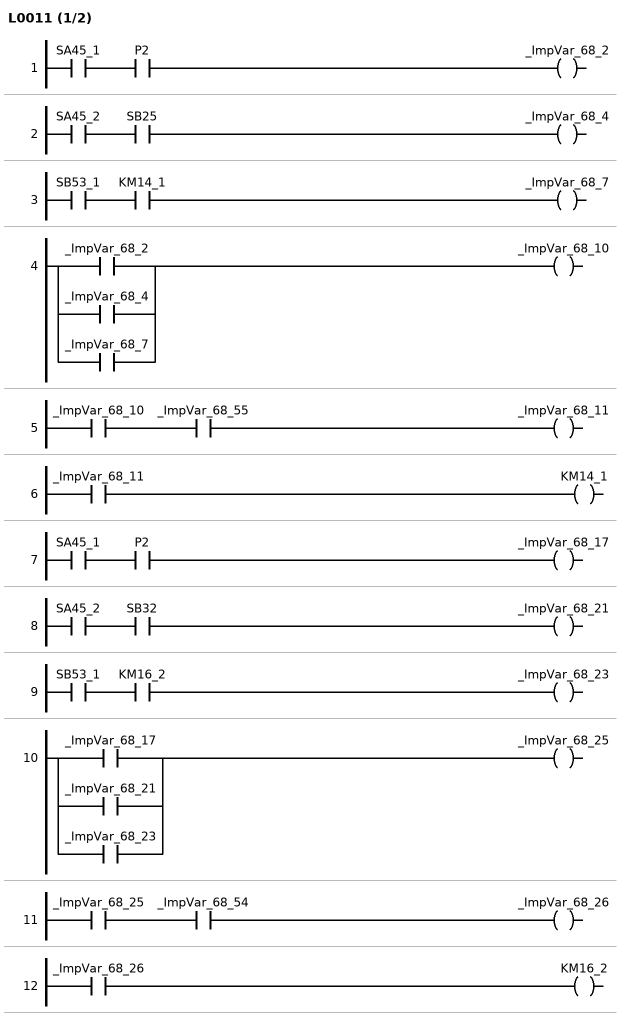
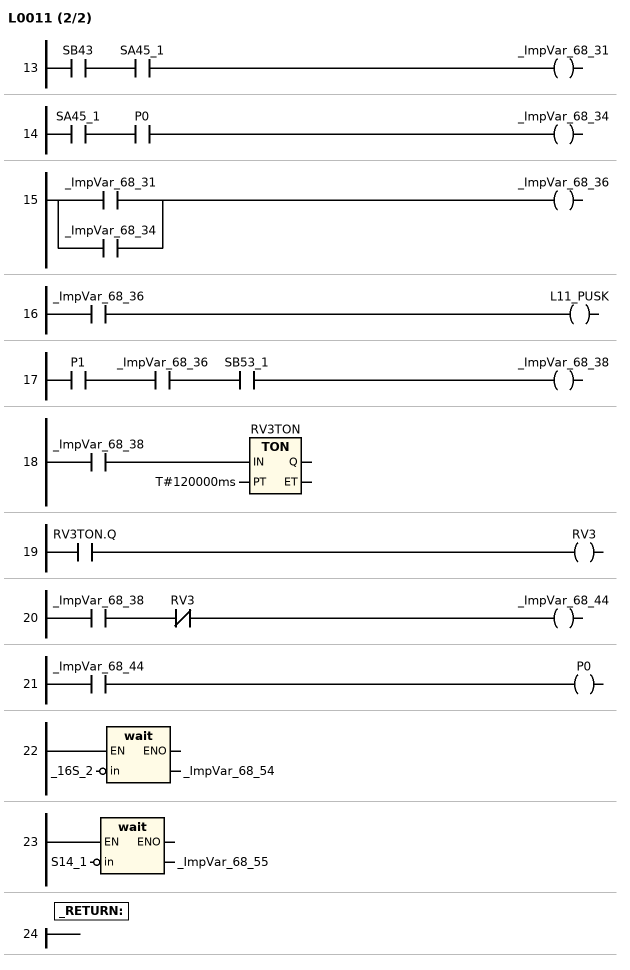
_LD_ (* Ladder Diagram *)
NETWORK 1
	[SA45_1] - [P2] --- (_ImpVar_68_2)
NETWORK 2
	[SA45_2] - [SB25] --- (_ImpVar_68_4)
NETWORK 3
	[SB53_1] - [KM14_1] --- (_ImpVar_68_7)
NETWORK 4
	{ [_ImpVar_68_2] | [_ImpVar_68_4] | [_ImpVar_68_7] } --- (_ImpVar_68_10)
NETWORK 5
	[_ImpVar_68_10] - [_ImpVar_68_55] --- (_ImpVar_68_11)
NETWORK 6
	[_ImpVar_68_11] --- (KM14_1)
NETWORK 7
	[SA45_1] - [P2] --- (_ImpVar_68_17)
NETWORK 8
	[SA45_2] - [SB32] --- (_ImpVar_68_21)
NETWORK 9
	[SB53_1] - [KM16_2] --- (_ImpVar_68_23)
NETWORK 10
	{ [_ImpVar_68_17] | [_ImpVar_68_21] | [_ImpVar_68_23] } --- (_ImpVar_68_25)
NETWORK 11
	[_ImpVar_68_25] - [_ImpVar_68_54] --- (_ImpVar_68_26)
NETWORK 12
	[_ImpVar_68_26] --- (KM16_2)
NETWORK 13
	[SB43] - [SA45_1] --- (_ImpVar_68_31)
NETWORK 14
	[SA45_1] - [P0] --- (_ImpVar_68_34)
NETWORK 15
	{ [_ImpVar_68_31] | [_ImpVar_68_34] } --- (_ImpVar_68_36)
NETWORK 16
	[_ImpVar_68_36] --- (L11_PUSK)
NETWORK 17
	[P1] - [_ImpVar_68_36] - [SB53_1] --- (_ImpVar_68_38)
NETWORK 18
	[_ImpVar_68_38] - RV3TON:TON(IN: *, PT: T#120000ms)
NETWORK 19
	[RV3TON.Q] --- (RV3)
NETWORK 20
	[_ImpVar_68_38] - [/RV3] --- (_ImpVar_68_44)
NETWORK 21
	[_ImpVar_68_44] --- (P0)
NETWORK 22
	*
		EN --- wait(in: NOT _16S_2) => _ImpVar_68_54
NETWORK 23
	*
		EN --- wait(in: NOT S14_1) => _ImpVar_68_55
NETWORK 24 _RETURN::
	*
_END_LD_
(* the same logic as Structured Text *)
(* Network 1 *)
_ImpVar_68_2 := SA45_1 AND P2;
(* Network 2 *)
_ImpVar_68_4 := SA45_2 AND SB25;
(* Network 3 *)
_ImpVar_68_7 := SB53_1 AND KM14_1;
(* Network 4 *)
_ImpVar_68_10 := _ImpVar_68_2 OR _ImpVar_68_4 OR _ImpVar_68_7;
(* Network 5 *)
_ImpVar_68_11 := _ImpVar_68_10 AND _ImpVar_68_55;
(* Network 6 *)
KM14_1 := _ImpVar_68_11;
(* Network 7 *)
_ImpVar_68_17 := SA45_1 AND P2;
(* Network 8 *)
_ImpVar_68_21 := SA45_2 AND SB32;
(* Network 9 *)
_ImpVar_68_23 := SB53_1 AND KM16_2;
(* Network 10 *)
_ImpVar_68_25 := _ImpVar_68_17 OR _ImpVar_68_21 OR _ImpVar_68_23;
(* Network 11 *)
_ImpVar_68_26 := _ImpVar_68_25 AND _ImpVar_68_54;
(* Network 12 *)
KM16_2 := _ImpVar_68_26;
(* Network 13 *)
_ImpVar_68_31 := SB43 AND SA45_1;
(* Network 14 *)
_ImpVar_68_34 := SA45_1 AND P0;
(* Network 15 *)
_ImpVar_68_36 := _ImpVar_68_31 OR _ImpVar_68_34;
(* Network 16 *)
L11_PUSK := _ImpVar_68_36;
(* Network 17 *)
_ImpVar_68_38 := P1 AND _ImpVar_68_36 AND SB53_1;
(* Network 18 *)
RV3TON(IN := _ImpVar_68_38, PT := T#120000ms);
(* Network 19 *)
RV3 := RV3TON.Q;
(* Network 20 *)
_ImpVar_68_44 := _ImpVar_68_38 AND NOT RV3;
(* Network 21 *)
P0 := _ImpVar_68_44;
(* Network 22 *)
_ImpVar_68_54 := wait(in := NOT _16S_2);
(* Network 23 *)
_ImpVar_68_55 := wait(in := NOT S14_1);
(* Network 24 *)
(* label: _RETURN: *)
END_PROGRAM

(* POU L0012, LD *)
PROGRAM L0012
VAR







END_VAR
VAR
	_ImpVar_72_9:	BOOL;
	_ImpVar_72_4:	BOOL;
	_ImpVar_72_7:	BOOL;
	_ImpVar_72_12:	BOOL;
	_ImpVar_72_5:	BOOL;
	_ImpVar_72_15:	BOOL;
	_ImpVar_72_20:	BOOL;
	_ImpVar_72_33:	BOOL;
	_ImpVar_72_22:	BOOL;
	_ImpVar_72_25:	BOOL;
	_ImpVar_72_27:	BOOL;
	_ImpVar_72_35:	BOOL;
	_ImpVar_72_38:	BOOL;
	_ImpVar_72_41:	BOOL;
	_ImpVar_72_45:	BOOL;
	_ImpVar_72_46:	BOOL;
	_ImpVar_72_52:	BOOL;
	_ImpVar_72_54:	BOOL;
	_ImpVar_72_56:	BOOL;
	_ImpVar_72_59:	BOOL;
	_ImpVar_72_60:	BOOL;
	_ImpVar_72_85:	BOOL;
	_ImpVar_72_86:	BOOL;
	_ImpVar_72_87:	BOOL;
	_ImpVar_72_88:	BOOL;

END_VAR
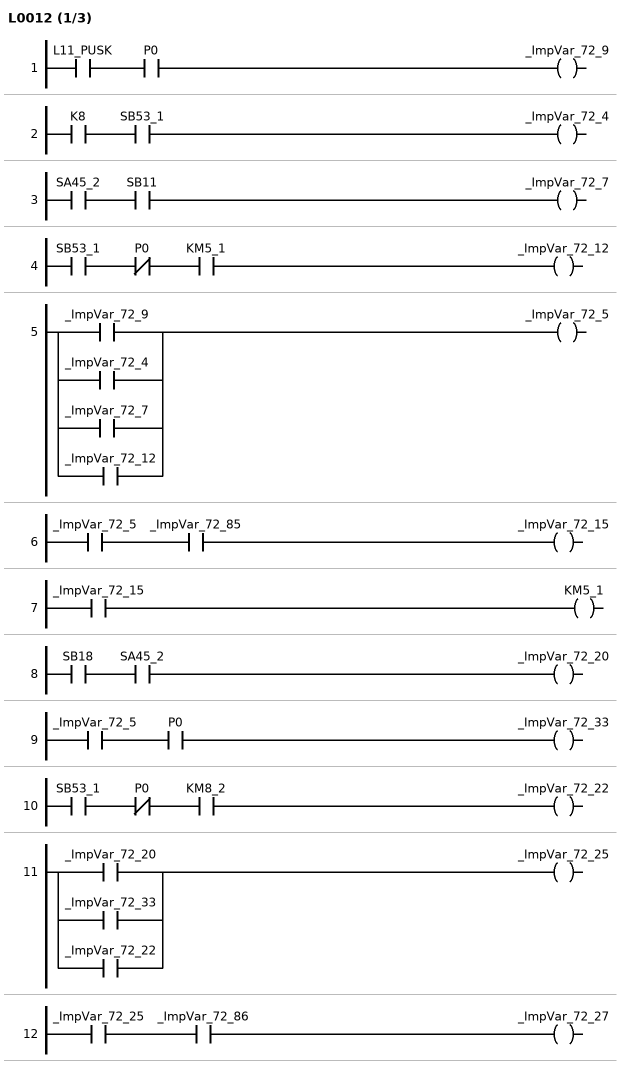
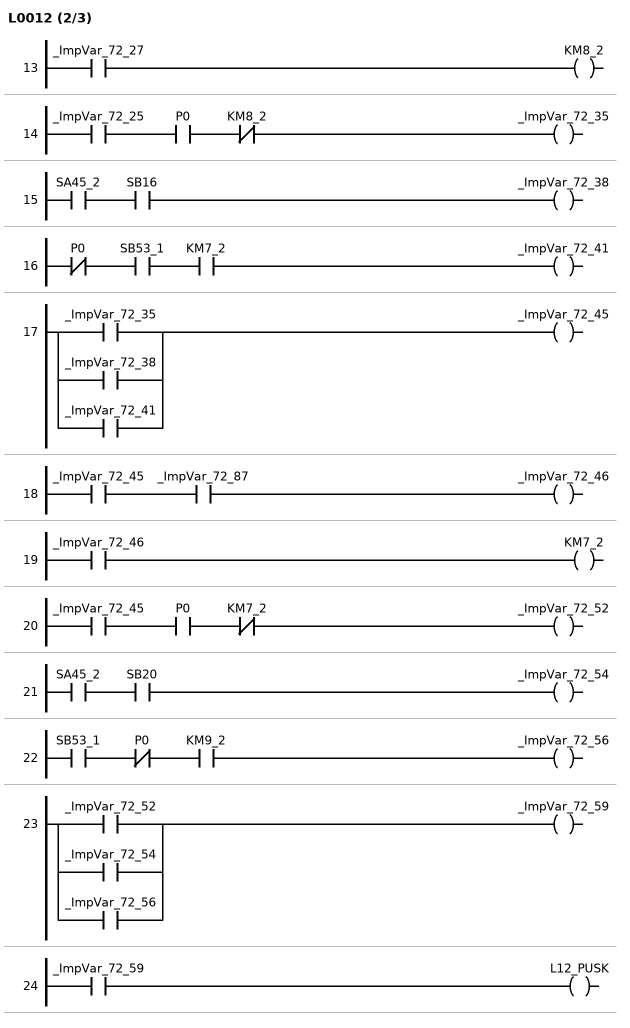
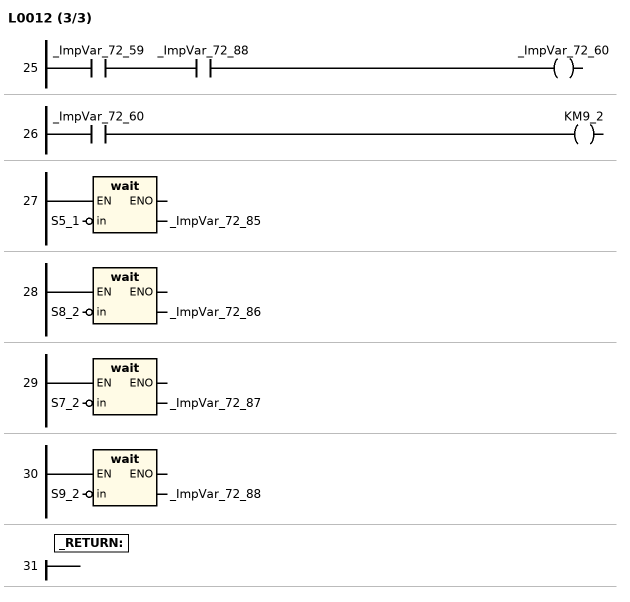
_LD_ (* Ladder Diagram *)
NETWORK 1
	[L11_PUSK] - [P0] --- (_ImpVar_72_9)
NETWORK 2
	[K8] - [SB53_1] --- (_ImpVar_72_4)
NETWORK 3
	[SA45_2] - [SB11] --- (_ImpVar_72_7)
NETWORK 4
	[SB53_1] - [/P0] - [KM5_1] --- (_ImpVar_72_12)
NETWORK 5
	{ [_ImpVar_72_9] | [_ImpVar_72_4] | [_ImpVar_72_7] | [_ImpVar_72_12] } --- (_ImpVar_72_5)
NETWORK 6
	[_ImpVar_72_5] - [_ImpVar_72_85] --- (_ImpVar_72_15)
NETWORK 7
	[_ImpVar_72_15] --- (KM5_1)
NETWORK 8
	[SB18] - [SA45_2] --- (_ImpVar_72_20)
NETWORK 9
	[_ImpVar_72_5] - [P0] --- (_ImpVar_72_33)
NETWORK 10
	[SB53_1] - [/P0] - [KM8_2] --- (_ImpVar_72_22)
NETWORK 11
	{ [_ImpVar_72_20] | [_ImpVar_72_33] | [_ImpVar_72_22] } --- (_ImpVar_72_25)
NETWORK 12
	[_ImpVar_72_25] - [_ImpVar_72_86] --- (_ImpVar_72_27)
NETWORK 13
	[_ImpVar_72_27] --- (KM8_2)
NETWORK 14
	[_ImpVar_72_25] - [P0] - [/KM8_2] --- (_ImpVar_72_35)
NETWORK 15
	[SA45_2] - [SB16] --- (_ImpVar_72_38)
NETWORK 16
	[/P0] - [SB53_1] - [KM7_2] --- (_ImpVar_72_41)
NETWORK 17
	{ [_ImpVar_72_35] | [_ImpVar_72_38] | [_ImpVar_72_41] } --- (_ImpVar_72_45)
NETWORK 18
	[_ImpVar_72_45] - [_ImpVar_72_87] --- (_ImpVar_72_46)
NETWORK 19
	[_ImpVar_72_46] --- (KM7_2)
NETWORK 20
	[_ImpVar_72_45] - [P0] - [/KM7_2] --- (_ImpVar_72_52)
NETWORK 21
	[SA45_2] - [SB20] --- (_ImpVar_72_54)
NETWORK 22
	[SB53_1] - [/P0] - [KM9_2] --- (_ImpVar_72_56)
NETWORK 23
	{ [_ImpVar_72_52] | [_ImpVar_72_54] | [_ImpVar_72_56] } --- (_ImpVar_72_59)
NETWORK 24
	[_ImpVar_72_59] --- (L12_PUSK)
NETWORK 25
	[_ImpVar_72_59] - [_ImpVar_72_88] --- (_ImpVar_72_60)
NETWORK 26
	[_ImpVar_72_60] --- (KM9_2)
NETWORK 27
	*
		EN --- wait(in: NOT S5_1) => _ImpVar_72_85
NETWORK 28
	*
		EN --- wait(in: NOT S8_2) => _ImpVar_72_86
NETWORK 29
	*
		EN --- wait(in: NOT S7_2) => _ImpVar_72_87
NETWORK 30
	*
		EN --- wait(in: NOT S9_2) => _ImpVar_72_88
NETWORK 31 _RETURN::
	*
_END_LD_
(* the same logic as Structured Text *)
(* Network 1 *)
_ImpVar_72_9 := L11_PUSK AND P0;
(* Network 2 *)
_ImpVar_72_4 := K8 AND SB53_1;
(* Network 3 *)
_ImpVar_72_7 := SA45_2 AND SB11;
(* Network 4 *)
_ImpVar_72_12 := SB53_1 AND NOT P0 AND KM5_1;
(* Network 5 *)
_ImpVar_72_5 := _ImpVar_72_9 OR _ImpVar_72_4 OR _ImpVar_72_7 OR _ImpVar_72_12;
(* Network 6 *)
_ImpVar_72_15 := _ImpVar_72_5 AND _ImpVar_72_85;
(* Network 7 *)
KM5_1 := _ImpVar_72_15;
(* Network 8 *)
_ImpVar_72_20 := SB18 AND SA45_2;
(* Network 9 *)
_ImpVar_72_33 := _ImpVar_72_5 AND P0;
(* Network 10 *)
_ImpVar_72_22 := SB53_1 AND NOT P0 AND KM8_2;
(* Network 11 *)
_ImpVar_72_25 := _ImpVar_72_20 OR _ImpVar_72_33 OR _ImpVar_72_22;
(* Network 12 *)
_ImpVar_72_27 := _ImpVar_72_25 AND _ImpVar_72_86;
(* Network 13 *)
KM8_2 := _ImpVar_72_27;
(* Network 14 *)
_ImpVar_72_35 := _ImpVar_72_25 AND P0 AND NOT KM8_2;
(* Network 15 *)
_ImpVar_72_38 := SA45_2 AND SB16;
(* Network 16 *)
_ImpVar_72_41 := NOT P0 AND SB53_1 AND KM7_2;
(* Network 17 *)
_ImpVar_72_45 := _ImpVar_72_35 OR _ImpVar_72_38 OR _ImpVar_72_41;
(* Network 18 *)
_ImpVar_72_46 := _ImpVar_72_45 AND _ImpVar_72_87;
(* Network 19 *)
KM7_2 := _ImpVar_72_46;
(* Network 20 *)
_ImpVar_72_52 := _ImpVar_72_45 AND P0 AND NOT KM7_2;
(* Network 21 *)
_ImpVar_72_54 := SA45_2 AND SB20;
(* Network 22 *)
_ImpVar_72_56 := SB53_1 AND NOT P0 AND KM9_2;
(* Network 23 *)
_ImpVar_72_59 := _ImpVar_72_52 OR _ImpVar_72_54 OR _ImpVar_72_56;
(* Network 24 *)
L12_PUSK := _ImpVar_72_59;
(* Network 25 *)
_ImpVar_72_60 := _ImpVar_72_59 AND _ImpVar_72_88;
(* Network 26 *)
KM9_2 := _ImpVar_72_60;
(* Network 27 *)
_ImpVar_72_85 := wait(in := NOT S5_1);
(* Network 28 *)
_ImpVar_72_86 := wait(in := NOT S8_2);
(* Network 29 *)
_ImpVar_72_87 := wait(in := NOT S7_2);
(* Network 30 *)
_ImpVar_72_88 := wait(in := NOT S9_2);
(* Network 31 *)
(* label: _RETURN: *)
END_PROGRAM

(* POU L0013, LD *)
PROGRAM L0013
VAR



	P4: BOOL;

END_VAR
VAR
	_ImpVar_78_4:	BOOL;
	_ImpVar_78_7:	BOOL;
	_ImpVar_78_11:	BOOL;
	_ImpVar_78_12:	BOOL;
	_ImpVar_78_42:	BOOL;
	_ImpVar_78_13:	BOOL;
	_ImpVar_78_20:	BOOL;
	_ImpVar_78_19:	BOOL;
	_ImpVar_78_23:	BOOL;
	_ImpVar_78_43:	BOOL;
	_ImpVar_78_26:	BOOL;
	_ImpVar_78_31:	BOOL;
	_ImpVar_78_32:	BOOL;

END_VAR
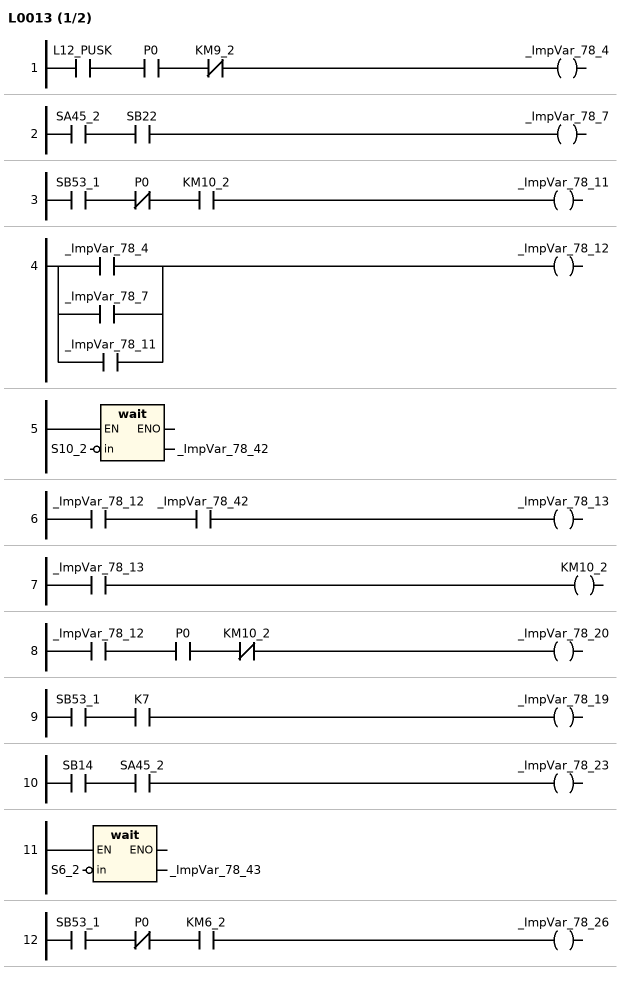
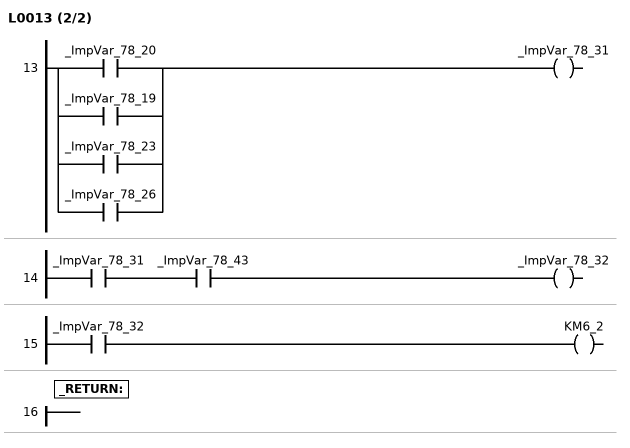
_LD_ (* Ladder Diagram *)
NETWORK 1
	[L12_PUSK] - [P0] - [/KM9_2] --- (_ImpVar_78_4)
NETWORK 2
	[SA45_2] - [SB22] --- (_ImpVar_78_7)
NETWORK 3
	[SB53_1] - [/P0] - [KM10_2] --- (_ImpVar_78_11)
NETWORK 4
	{ [_ImpVar_78_4] | [_ImpVar_78_7] | [_ImpVar_78_11] } --- (_ImpVar_78_12)
NETWORK 5
	*
		EN --- wait(in: NOT S10_2) => _ImpVar_78_42
NETWORK 6
	[_ImpVar_78_12] - [_ImpVar_78_42] --- (_ImpVar_78_13)
NETWORK 7
	[_ImpVar_78_13] --- (KM10_2)
NETWORK 8
	[_ImpVar_78_12] - [P0] - [/KM10_2] --- (_ImpVar_78_20)
NETWORK 9
	[SB53_1] - [K7] --- (_ImpVar_78_19)
NETWORK 10
	[SB14] - [SA45_2] --- (_ImpVar_78_23)
NETWORK 11
	*
		EN --- wait(in: NOT S6_2) => _ImpVar_78_43
NETWORK 12
	[SB53_1] - [/P0] - [KM6_2] --- (_ImpVar_78_26)
NETWORK 13
	{ [_ImpVar_78_20] | [_ImpVar_78_19] | [_ImpVar_78_23] | [_ImpVar_78_26] } --- (_ImpVar_78_31)
NETWORK 14
	[_ImpVar_78_31] - [_ImpVar_78_43] --- (_ImpVar_78_32)
NETWORK 15
	[_ImpVar_78_32] --- (KM6_2)
NETWORK 16 _RETURN::
	*
_END_LD_
(* the same logic as Structured Text *)
(* Network 1 *)
_ImpVar_78_4 := L12_PUSK AND P0 AND NOT KM9_2;
(* Network 2 *)
_ImpVar_78_7 := SA45_2 AND SB22;
(* Network 3 *)
_ImpVar_78_11 := SB53_1 AND NOT P0 AND KM10_2;
(* Network 4 *)
_ImpVar_78_12 := _ImpVar_78_4 OR _ImpVar_78_7 OR _ImpVar_78_11;
(* Network 5 *)
_ImpVar_78_42 := wait(in := NOT S10_2);
(* Network 6 *)
_ImpVar_78_13 := _ImpVar_78_12 AND _ImpVar_78_42;
(* Network 7 *)
KM10_2 := _ImpVar_78_13;
(* Network 8 *)
_ImpVar_78_20 := _ImpVar_78_12 AND P0 AND NOT KM10_2;
(* Network 9 *)
_ImpVar_78_19 := SB53_1 AND K7;
(* Network 10 *)
_ImpVar_78_23 := SB14 AND SA45_2;
(* Network 11 *)
_ImpVar_78_43 := wait(in := NOT S6_2);
(* Network 12 *)
_ImpVar_78_26 := SB53_1 AND NOT P0 AND KM6_2;
(* Network 13 *)
_ImpVar_78_31 := _ImpVar_78_20 OR _ImpVar_78_19 OR _ImpVar_78_23 OR _ImpVar_78_26;
(* Network 14 *)
_ImpVar_78_32 := _ImpVar_78_31 AND _ImpVar_78_43;
(* Network 15 *)
KM6_2 := _ImpVar_78_32;
(* Network 16 *)
(* label: _RETURN: *)
END_PROGRAM

(* POU L0014, LD *)
PROGRAM L0014
VAR

END_VAR
VAR
	_ImpVar_83_6:	BOOL;
	_ImpVar_83_56:	BOOL;
	_ImpVar_83_9:	BOOL;
	_ImpVar_83_12:	BOOL;
	_ImpVar_83_13:	BOOL;
	_ImpVar_83_24:	BOOL;
	_ImpVar_83_27:	BOOL;
	_ImpVar_83_29:	BOOL;
	_ImpVar_83_57:	BOOL;
	_ImpVar_83_30:	BOOL;

END_VAR
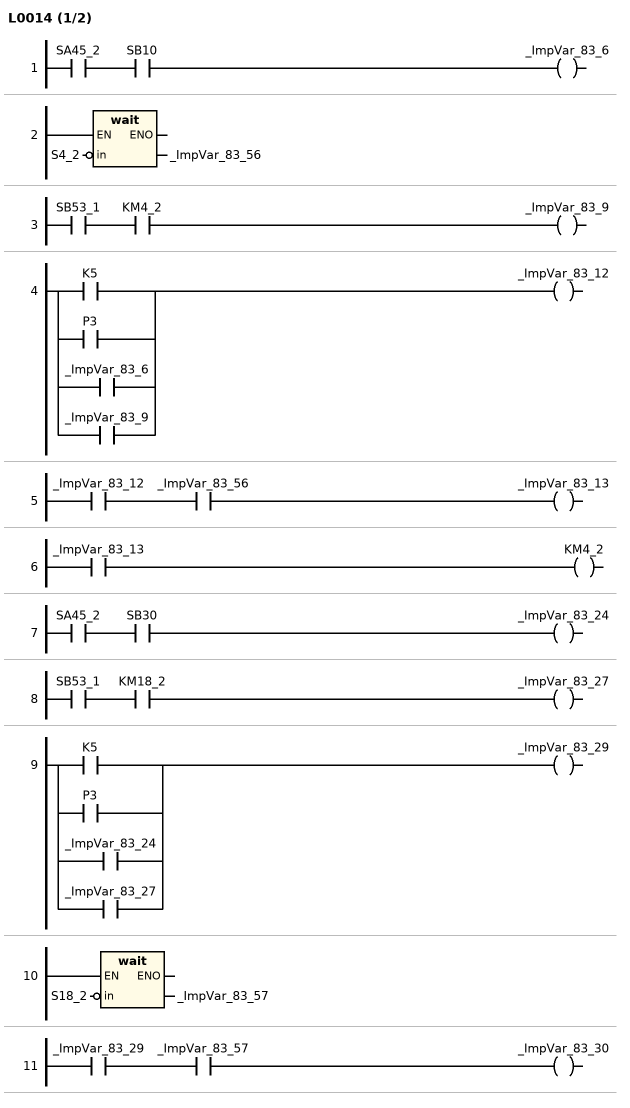
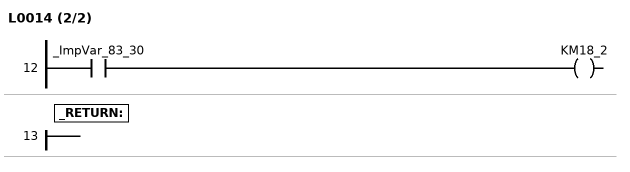
_LD_ (* Ladder Diagram *)
NETWORK 1
	[SA45_2] - [SB10] --- (_ImpVar_83_6)
NETWORK 2
	*
		EN --- wait(in: NOT S4_2) => _ImpVar_83_56
NETWORK 3
	[SB53_1] - [KM4_2] --- (_ImpVar_83_9)
NETWORK 4
	{ [K5] | [P3] | [_ImpVar_83_6] | [_ImpVar_83_9] } --- (_ImpVar_83_12)
NETWORK 5
	[_ImpVar_83_12] - [_ImpVar_83_56] --- (_ImpVar_83_13)
NETWORK 6
	[_ImpVar_83_13] --- (KM4_2)
NETWORK 7
	[SA45_2] - [SB30] --- (_ImpVar_83_24)
NETWORK 8
	[SB53_1] - [KM18_2] --- (_ImpVar_83_27)
NETWORK 9
	{ [K5] | [P3] | [_ImpVar_83_24] | [_ImpVar_83_27] } --- (_ImpVar_83_29)
NETWORK 10
	*
		EN --- wait(in: NOT S18_2) => _ImpVar_83_57
NETWORK 11
	[_ImpVar_83_29] - [_ImpVar_83_57] --- (_ImpVar_83_30)
NETWORK 12
	[_ImpVar_83_30] --- (KM18_2)
NETWORK 13 _RETURN::
	*
_END_LD_
(* the same logic as Structured Text *)
(* Network 1 *)
_ImpVar_83_6 := SA45_2 AND SB10;
(* Network 2 *)
_ImpVar_83_56 := wait(in := NOT S4_2);
(* Network 3 *)
_ImpVar_83_9 := SB53_1 AND KM4_2;
(* Network 4 *)
_ImpVar_83_12 := K5 OR P3 OR _ImpVar_83_6 OR _ImpVar_83_9;
(* Network 5 *)
_ImpVar_83_13 := _ImpVar_83_12 AND _ImpVar_83_56;
(* Network 6 *)
KM4_2 := _ImpVar_83_13;
(* Network 7 *)
_ImpVar_83_24 := SA45_2 AND SB30;
(* Network 8 *)
_ImpVar_83_27 := SB53_1 AND KM18_2;
(* Network 9 *)
_ImpVar_83_29 := K5 OR P3 OR _ImpVar_83_24 OR _ImpVar_83_27;
(* Network 10 *)
_ImpVar_83_57 := wait(in := NOT S18_2);
(* Network 11 *)
_ImpVar_83_30 := _ImpVar_83_29 AND _ImpVar_83_57;
(* Network 12 *)
KM18_2 := _ImpVar_83_30;
(* Network 13 *)
(* label: _RETURN: *)
END_PROGRAM

(* POU L0015, LD *)
PROGRAM L0015
VAR

END_VAR
VAR
	_ImpVar_84_5:	BOOL;
	_ImpVar_84_11:	BOOL;
	_ImpVar_84_14:	BOOL;
	_ImpVar_84_56:	BOOL;
	_ImpVar_84_15:	BOOL;
	_ImpVar_84_20:	BOOL;
	_ImpVar_84_28:	BOOL;
	_ImpVar_84_34:	BOOL;
	_ImpVar_84_55:	BOOL;
	_ImpVar_84_21:	BOOL;
	_ImpVar_84_23:	BOOL;
	_ImpVar_84_46:	BOOL;
	_ImpVar_84_57:	BOOL;
	_ImpVar_84_52:	BOOL;
	_ImpVar_84_39:	BOOL;
	_ImpVar_84_41:	BOOL;

END_VAR
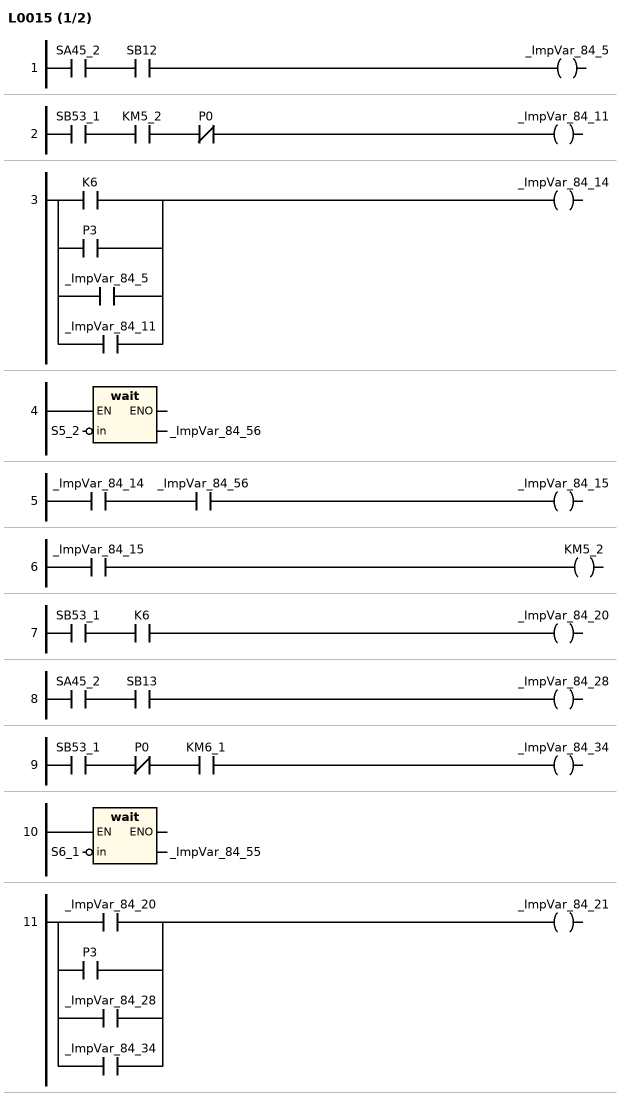
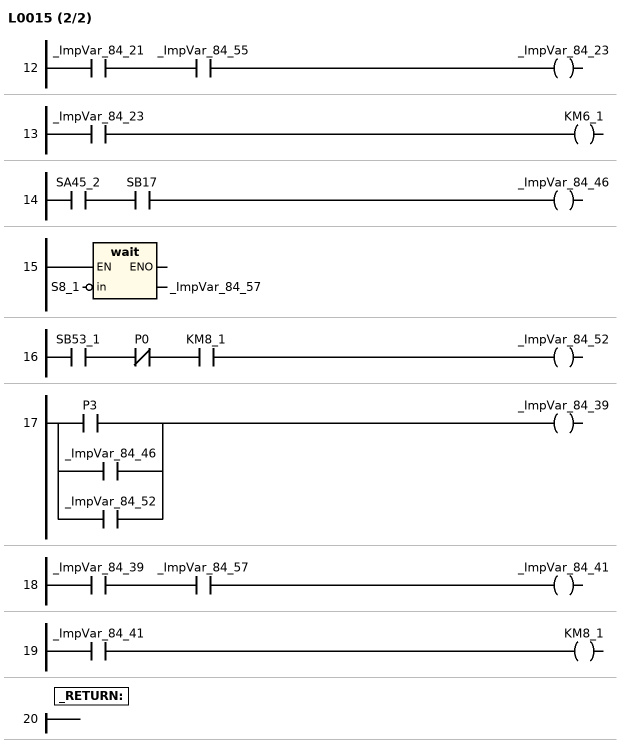
_LD_ (* Ladder Diagram *)
NETWORK 1
	[SA45_2] - [SB12] --- (_ImpVar_84_5)
NETWORK 2
	[SB53_1] - [KM5_2] - [/P0] --- (_ImpVar_84_11)
NETWORK 3
	{ [K6] | [P3] | [_ImpVar_84_5] | [_ImpVar_84_11] } --- (_ImpVar_84_14)
NETWORK 4
	*
		EN --- wait(in: NOT S5_2) => _ImpVar_84_56
NETWORK 5
	[_ImpVar_84_14] - [_ImpVar_84_56] --- (_ImpVar_84_15)
NETWORK 6
	[_ImpVar_84_15] --- (KM5_2)
NETWORK 7
	[SB53_1] - [K6] --- (_ImpVar_84_20)
NETWORK 8
	[SA45_2] - [SB13] --- (_ImpVar_84_28)
NETWORK 9
	[SB53_1] - [/P0] - [KM6_1] --- (_ImpVar_84_34)
NETWORK 10
	*
		EN --- wait(in: NOT S6_1) => _ImpVar_84_55
NETWORK 11
	{ [_ImpVar_84_20] | [P3] | [_ImpVar_84_28] | [_ImpVar_84_34] } --- (_ImpVar_84_21)
NETWORK 12
	[_ImpVar_84_21] - [_ImpVar_84_55] --- (_ImpVar_84_23)
NETWORK 13
	[_ImpVar_84_23] --- (KM6_1)
NETWORK 14
	[SA45_2] - [SB17] --- (_ImpVar_84_46)
NETWORK 15
	*
		EN --- wait(in: NOT S8_1) => _ImpVar_84_57
NETWORK 16
	[SB53_1] - [/P0] - [KM8_1] --- (_ImpVar_84_52)
NETWORK 17
	{ [P3] | [_ImpVar_84_46] | [_ImpVar_84_52] } --- (_ImpVar_84_39)
NETWORK 18
	[_ImpVar_84_39] - [_ImpVar_84_57] --- (_ImpVar_84_41)
NETWORK 19
	[_ImpVar_84_41] --- (KM8_1)
NETWORK 20 _RETURN::
	*
_END_LD_
(* the same logic as Structured Text *)
(* Network 1 *)
_ImpVar_84_5 := SA45_2 AND SB12;
(* Network 2 *)
_ImpVar_84_11 := SB53_1 AND KM5_2 AND NOT P0;
(* Network 3 *)
_ImpVar_84_14 := K6 OR P3 OR _ImpVar_84_5 OR _ImpVar_84_11;
(* Network 4 *)
_ImpVar_84_56 := wait(in := NOT S5_2);
(* Network 5 *)
_ImpVar_84_15 := _ImpVar_84_14 AND _ImpVar_84_56;
(* Network 6 *)
KM5_2 := _ImpVar_84_15;
(* Network 7 *)
_ImpVar_84_20 := SB53_1 AND K6;
(* Network 8 *)
_ImpVar_84_28 := SA45_2 AND SB13;
(* Network 9 *)
_ImpVar_84_34 := SB53_1 AND NOT P0 AND KM6_1;
(* Network 10 *)
_ImpVar_84_55 := wait(in := NOT S6_1);
(* Network 11 *)
_ImpVar_84_21 := _ImpVar_84_20 OR P3 OR _ImpVar_84_28 OR _ImpVar_84_34;
(* Network 12 *)
_ImpVar_84_23 := _ImpVar_84_21 AND _ImpVar_84_55;
(* Network 13 *)
KM6_1 := _ImpVar_84_23;
(* Network 14 *)
_ImpVar_84_46 := SA45_2 AND SB17;
(* Network 15 *)
_ImpVar_84_57 := wait(in := NOT S8_1);
(* Network 16 *)
_ImpVar_84_52 := SB53_1 AND NOT P0 AND KM8_1;
(* Network 17 *)
_ImpVar_84_39 := P3 OR _ImpVar_84_46 OR _ImpVar_84_52;
(* Network 18 *)
_ImpVar_84_41 := _ImpVar_84_39 AND _ImpVar_84_57;
(* Network 19 *)
KM8_1 := _ImpVar_84_41;
(* Network 20 *)
(* label: _RETURN: *)
END_PROGRAM

(* POU L0016, LD *)
PROGRAM L0016
VAR
	mt7TON: TON;

	mt9TON: TON;
	mt10TON: TON;
END_VAR
VAR
	_ImpVar_85_10:	BOOL;
	_ImpVar_85_16:	BOOL;
	_ImpVar_85_3:	BOOL;
	_ImpVar_85_130:	BOOL;
	_ImpVar_85_5:	BOOL;
	_ImpVar_85_57:	BOOL;
	_ImpVar_85_63:	BOOL;
	_ImpVar_85_51:	BOOL;
	_ImpVar_85_127:	BOOL;
	_ImpVar_85_52:	BOOL;
	_ImpVar_85_87:	BOOL;
	_ImpVar_85_93:	BOOL;
	_ImpVar_85_81:	BOOL;
	_ImpVar_85_128:	BOOL;
	_ImpVar_85_82:	BOOL;
	_ImpVar_85_102:	BOOL;
	_ImpVar_85_108:	BOOL;
	_ImpVar_85_96:	BOOL;
	_ImpVar_85_129:	BOOL;
	_ImpVar_85_97:	BOOL;
	_ImpVar_85_117:	BOOL;
	_ImpVar_85_123:	BOOL;
	_ImpVar_85_126:	BOOL;
	_ImpVar_85_131:	BOOL;
	_ImpVar_85_112:	BOOL;

END_VAR
